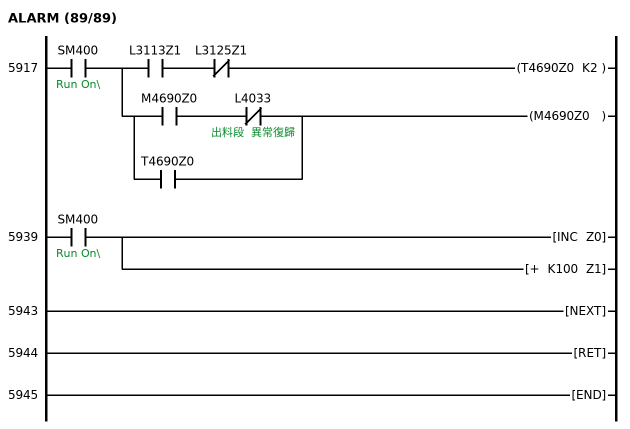
[picture p264: ladder of ALARM, rungs at steps 5917 to 5945]
5917  LD      SM400  ; Run On\
      MPS
      AND     L3113Z1
      ANI     L3125Z1
      OUT     T4690Z0 K2
      MPP
      LD      M4690Z0
      ANI     L4033  ; 出料段  異常復歸
      OR      T4690Z0
      ANB
      OUT     M4690Z0
5939  LD      SM400  ; Run On\
      INC     Z0
      +       K100 Z1
5943  NEXT
5944  RET
5945  END
END_PROGRAM

PROGRAM CCD_RB
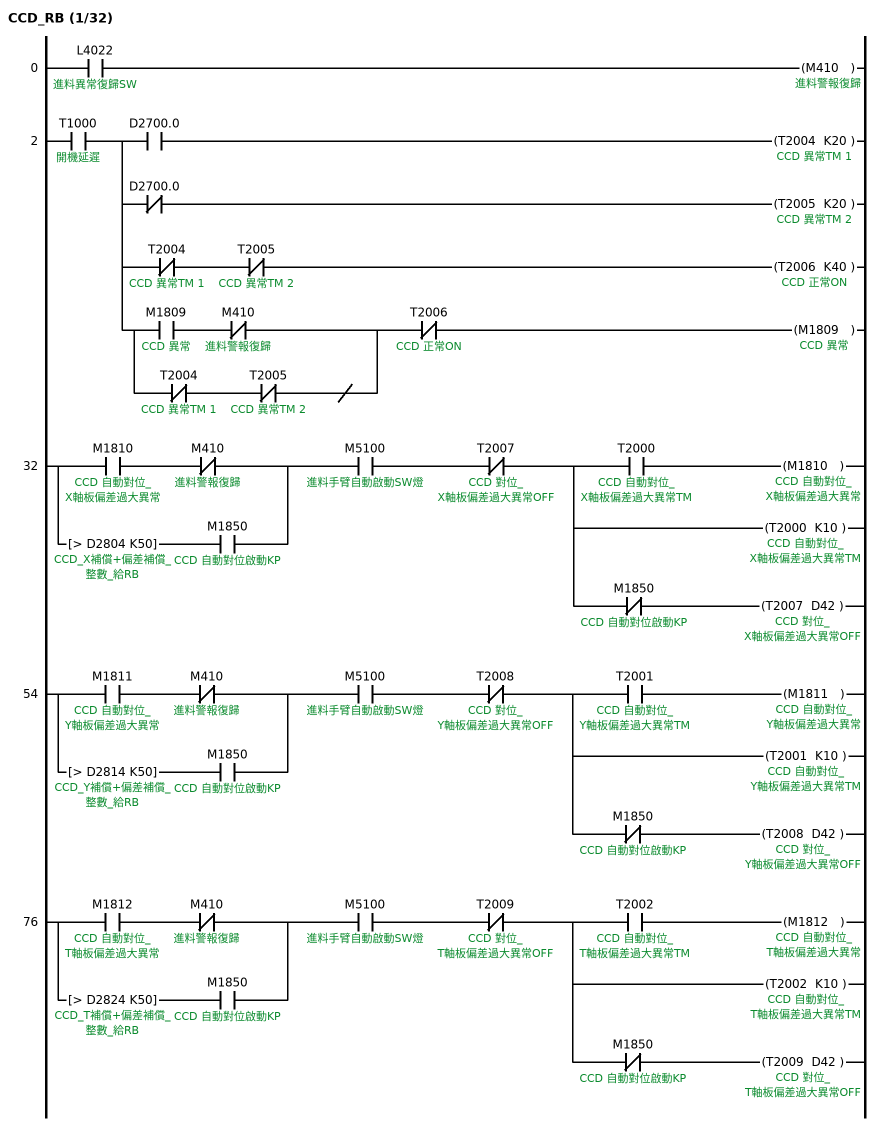
0     LD      L4022  ; 進料異常復歸SW
      OUT     M410  ; 進料警報復歸
2     LD      T1000  ; 開機延遲
      MPS
      AND     D2700.0
      OUT     T2004 K20  ; CCD 異常TM 1
      MRD
      ANI     D2700.0
      OUT     T2005 K20  ; CCD 異常TM 2
      MRD
      ANI     T2004  ; CCD 異常TM 1
      ANI     T2005  ; CCD 異常TM 2
      OUT     T2006 K40  ; CCD 正常ON
      MPP
      LD      M1809  ; CCD 異常
      ANI     M410  ; 進料警報復歸
      LDI     T2004  ; CCD 異常TM 1
      ANI     T2005  ; CCD 異常TM 2
      INV
      ORB
      ANB
      ANI     T2006  ; CCD 正常ON
      OUT     M1809  ; CCD 異常
32    LD      M1810  ; CCD 自動對位_X軸板偏差過大異常
      ANI     M410  ; 進料警報復歸
      LD>     D2804 K50  ; CCD_X補償+偏差補償_整數_給RB
      AND     M1850  ; CCD 自動對位啟動KP
      ORB
      AND     M5100  ; 進料手臂自動啟動SW燈
      ANI     T2007  ; CCD 對位_X軸板偏差過大異常OFF
      MPS
      AND     T2000  ; CCD 自動對位_X軸板偏差過大異常TM
      OUT     M1810  ; CCD 自動對位_X軸板偏差過大異常
      MPP
      OUT     T2000 K10  ; CCD 自動對位_X軸板偏差過大異常TM
      ANI     M1850  ; CCD 自動對位啟動KP
      OUT     T2007 D42  ; CCD 對位_X軸板偏差過大異常OFF
54    LD      M1811  ; CCD 自動對位_Y軸板偏差過大異常
      ANI     M410  ; 進料警報復歸
      LD>     D2814 K50  ; CCD_Y補償+偏差補償_整數_給RB
      AND     M1850  ; CCD 自動對位啟動KP
      ORB
      AND     M5100  ; 進料手臂自動啟動SW燈
      ANI     T2008  ; CCD 對位_Y軸板偏差過大異常OFF
      MPS
      AND     T2001  ; CCD 自動對位_Y軸板偏差過大異常TM
      OUT     M1811  ; CCD 自動對位_Y軸板偏差過大異常
      MPP
      OUT     T2001 K10  ; CCD 自動對位_Y軸板偏差過大異常TM
      ANI     M1850  ; CCD 自動對位啟動KP
      OUT     T2008 D42  ; CCD 對位_Y軸板偏差過大異常OFF
76    LD      M1812  ; CCD 自動對位_T軸板偏差過大異常
      ANI     M410  ; 進料警報復歸
      LD>     D2824 K50  ; CCD_T補償+偏差補償_整數_給RB
      AND     M1850  ; CCD 自動對位啟動KP
      ORB
      AND     M5100  ; 進料手臂自動啟動SW燈
      ANI     T2009  ; CCD 對位_T軸板偏差過大異常OFF
      MPS
      AND     T2002  ; CCD 自動對位_T軸板偏差過大異常TM
      OUT     M1812  ; CCD 自動對位_T軸板偏差過大異常
      MPP
      OUT     T2002 K10  ; CCD 自動對位_T軸板偏差過大異常TM
      ANI     M1850  ; CCD 自動對位啟動KP
      OUT     T2009 D42  ; CCD 對位_T軸板偏差過大異常OFF
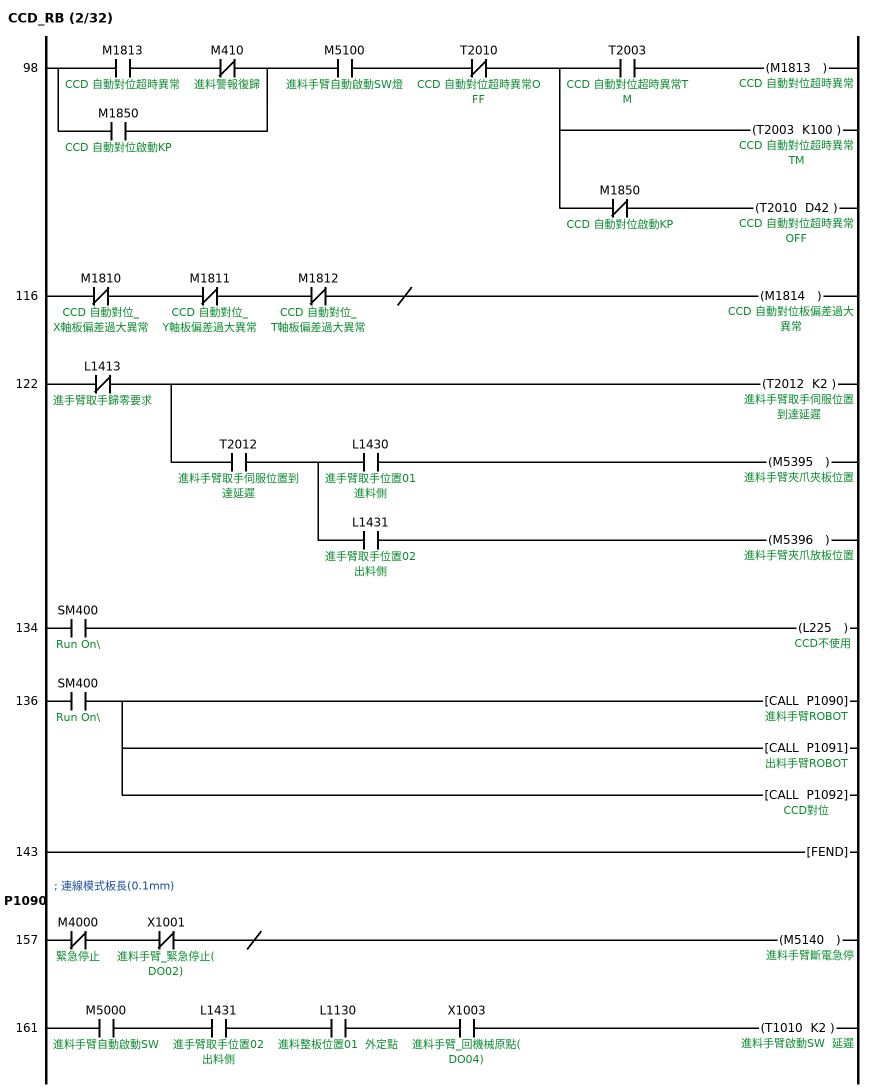
98    LD      M1813  ; CCD 自動對位超時異常
      ANI     M410  ; 進料警報復歸
      OR      M1850  ; CCD 自動對位啟動KP
      AND     M5100  ; 進料手臂自動啟動SW燈
      ANI     T2010  ; CCD 自動對位超時異常OFF
      MPS
      AND     T2003  ; CCD 自動對位超時異常TM
      OUT     M1813  ; CCD 自動對位超時異常
      MPP
      OUT     T2003 K100  ; CCD 自動對位超時異常TM
      ANI     M1850  ; CCD 自動對位啟動KP
      OUT     T2010 D42  ; CCD 自動對位超時異常OFF
116   LDI     M1810  ; CCD 自動對位_X軸板偏差過大異常
      ANI     M1811  ; CCD 自動對位_Y軸板偏差過大異常
      ANI     M1812  ; CCD 自動對位_T軸板偏差過大異常
      INV
      OUT     M1814  ; CCD 自動對位板偏差過大異常
122   LDI     L1413  ; 進手臂取手歸零要求
      OUT     T2012 K2  ; 進料手臂取手伺服位置到達延遲
      AND     T2012  ; 進料手臂取手伺服位置到達延遲
      MPS
      AND     L1430  ; 進手臂取手位置01  進料側
      OUT     M5395  ; 進料手臂夾爪夾板位置
      MPP
      AND     L1431  ; 進手臂取手位置02  出料側
      OUT     M5396  ; 進料手臂夾爪放板位置
134   LD      SM400  ; Run On\
      OUT     L225  ; CCD不使用
136   LD      SM400  ; Run On\
      CALL    P1090  ; 進料手臂ROBOT
      CALL    P1091  ; 出料手臂ROBOT
      CALL    P1092  ; CCD對位
143   FEND
; 連線模式板長(0.1mm)
      P1090
157   LDI     M4000  ; 緊急停止
      ANI     X1001  ; 進料手臂_緊急停止(DO02)
      INV
      OUT     M5140  ; 進料手臂斷電急停
161   LD      M5000  ; 進料手臂自動啟動SW
      AND     L1431  ; 進手臂取手位置02  出料側
      AND     L1130  ; 進料整板位置01  外定點
      AND     X1003  ; 進料手臂_回機械原點(DO04)
      OUT     T1010 K2  ; 進料手臂啟動SW  延遲
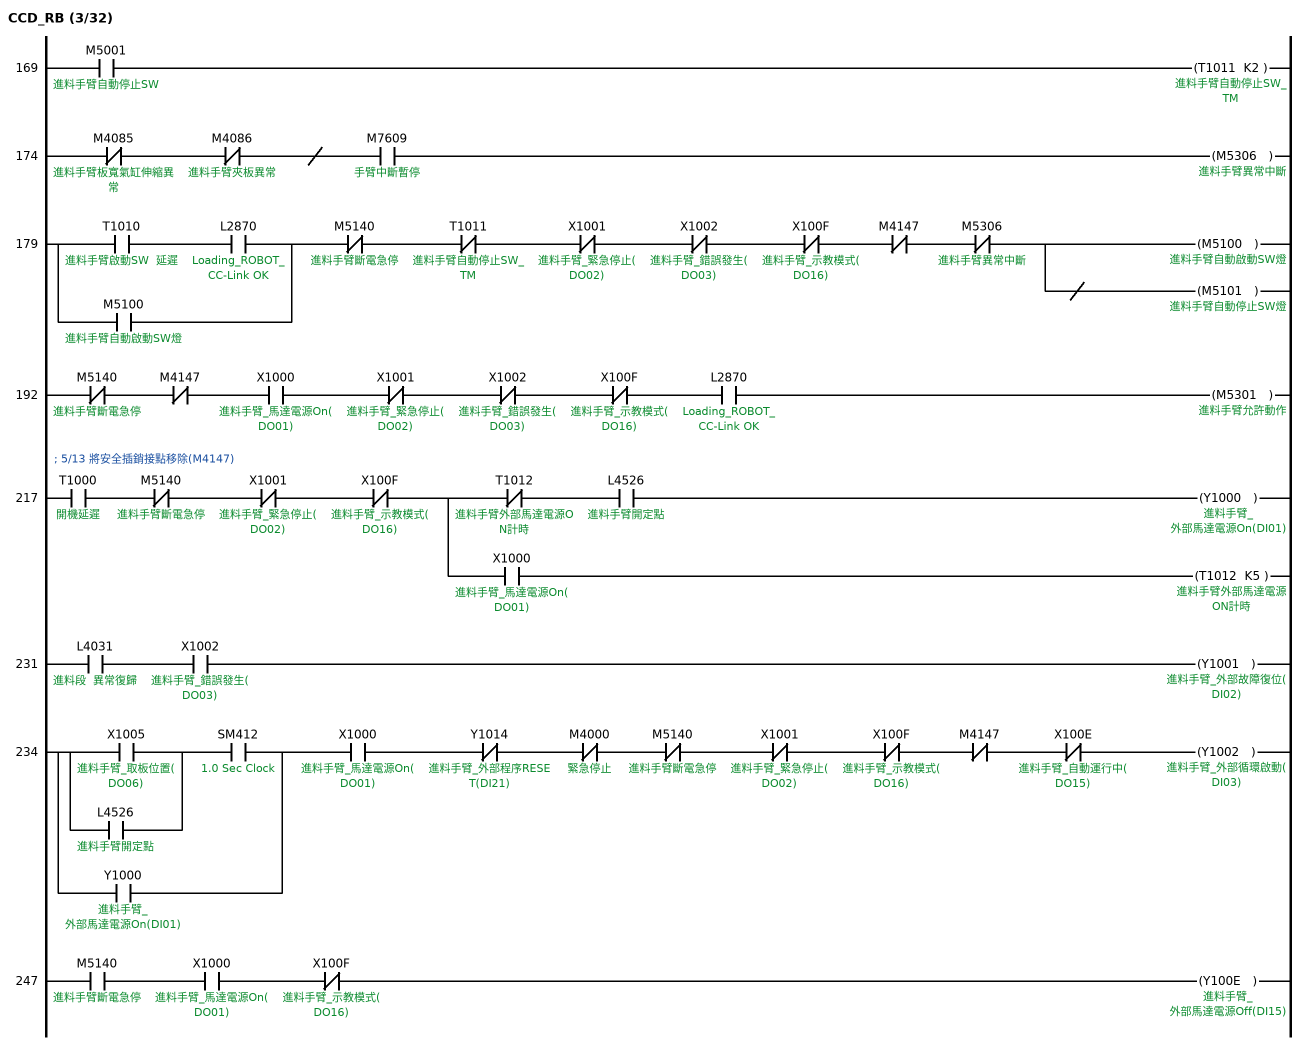
169   LD      M5001  ; 進料手臂自動停止SW
      OUT     T1011 K2  ; 進料手臂自動停止SW_TM
174   LDI     M4085  ; 進料手臂板寬氣缸伸縮異常
      ANI     M4086  ; 進料手臂夾板異常
      INV
      AND     M7609  ; 手臂中斷暫停
      OUT     M5306  ; 進料手臂異常中斷
179   LD      T1010  ; 進料手臂啟動SW  延遲
      AND     L2870  ; Loading_ROBOT_  CC-Link OK
      OR      M5100  ; 進料手臂自動啟動SW燈
      ANI     M5140  ; 進料手臂斷電急停
      ANI     T1011  ; 進料手臂自動停止SW_TM
      ANI     X1001  ; 進料手臂_緊急停止(DO02)
      ANI     X1002  ; 進料手臂_錯誤發生(DO03)
      ANI     X100F  ; 進料手臂_示教模式(DO16)
      ANI     M4147
      ANI     M5306  ; 進料手臂異常中斷
      OUT     M5100  ; 進料手臂自動啟動SW燈
      INV
      OUT     M5101  ; 進料手臂自動停止SW燈
192   LDI     M5140  ; 進料手臂斷電急停
      ANI     M4147
      AND     X1000  ; 進料手臂_馬達電源On(DO01)
      ANI     X1001  ; 進料手臂_緊急停止(DO02)
      ANI     X1002  ; 進料手臂_錯誤發生(DO03)
      ANI     X100F  ; 進料手臂_示教模式(DO16)
      AND     L2870  ; Loading_ROBOT_  CC-Link OK
      OUT     M5301  ; 進料手臂允許動作
; 5/13 將安全插銷接點移除(M4147)
217   LD      T1000  ; 開機延遲
      ANI     M5140  ; 進料手臂斷電急停
      ANI     X1001  ; 進料手臂_緊急停止(DO02)
      ANI     X100F  ; 進料手臂_示教模式(DO16)
      MPS
      ANI     T1012  ; 進料手臂外部馬達電源ON計時
      AND     L4526  ; 進料手臂開定點
      OUT     Y1000  ; 進料手臂_外部馬達電源On(DI01)
      MPP
      AND     X1000  ; 進料手臂_馬達電源On(DO01)
      OUT     T1012 K5  ; 進料手臂外部馬達電源ON計時
231   LD      L4031  ; 進料段  異常復歸
      AND     X1002  ; 進料手臂_錯誤發生(DO03)
      OUT     Y1001  ; 進料手臂_外部故障復位(DI02)
234   LD      X1005  ; 進料手臂_取板位置(DO06)
      OR      L4526  ; 進料手臂開定點
      AND     SM412  ; 1.0 Sec Clock
      OR      Y1000  ; 進料手臂_外部馬達電源On(DI01)
      AND     X1000  ; 進料手臂_馬達電源On(DO01)
      ANI     Y1014  ; 進料手臂_外部程序RESET(DI21)
      ANI     M4000  ; 緊急停止
      ANI     M5140  ; 進料手臂斷電急停
      ANI     X1001  ; 進料手臂_緊急停止(DO02)
      ANI     X100F  ; 進料手臂_示教模式(DO16)
      ANI     M4147
      ANI     X100E  ; 進料手臂_自動運行中(DO15)
      OUT     Y1002  ; 進料手臂_外部循環啟動(DI03)
247   LD      M5140  ; 進料手臂斷電急停
      AND     X1000  ; 進料手臂_馬達電源On(DO01)
      ANI     X100F  ; 進料手臂_示教模式(DO16)
      OUT     Y100E  ; 進料手臂_外部馬達電源Off(DI15)
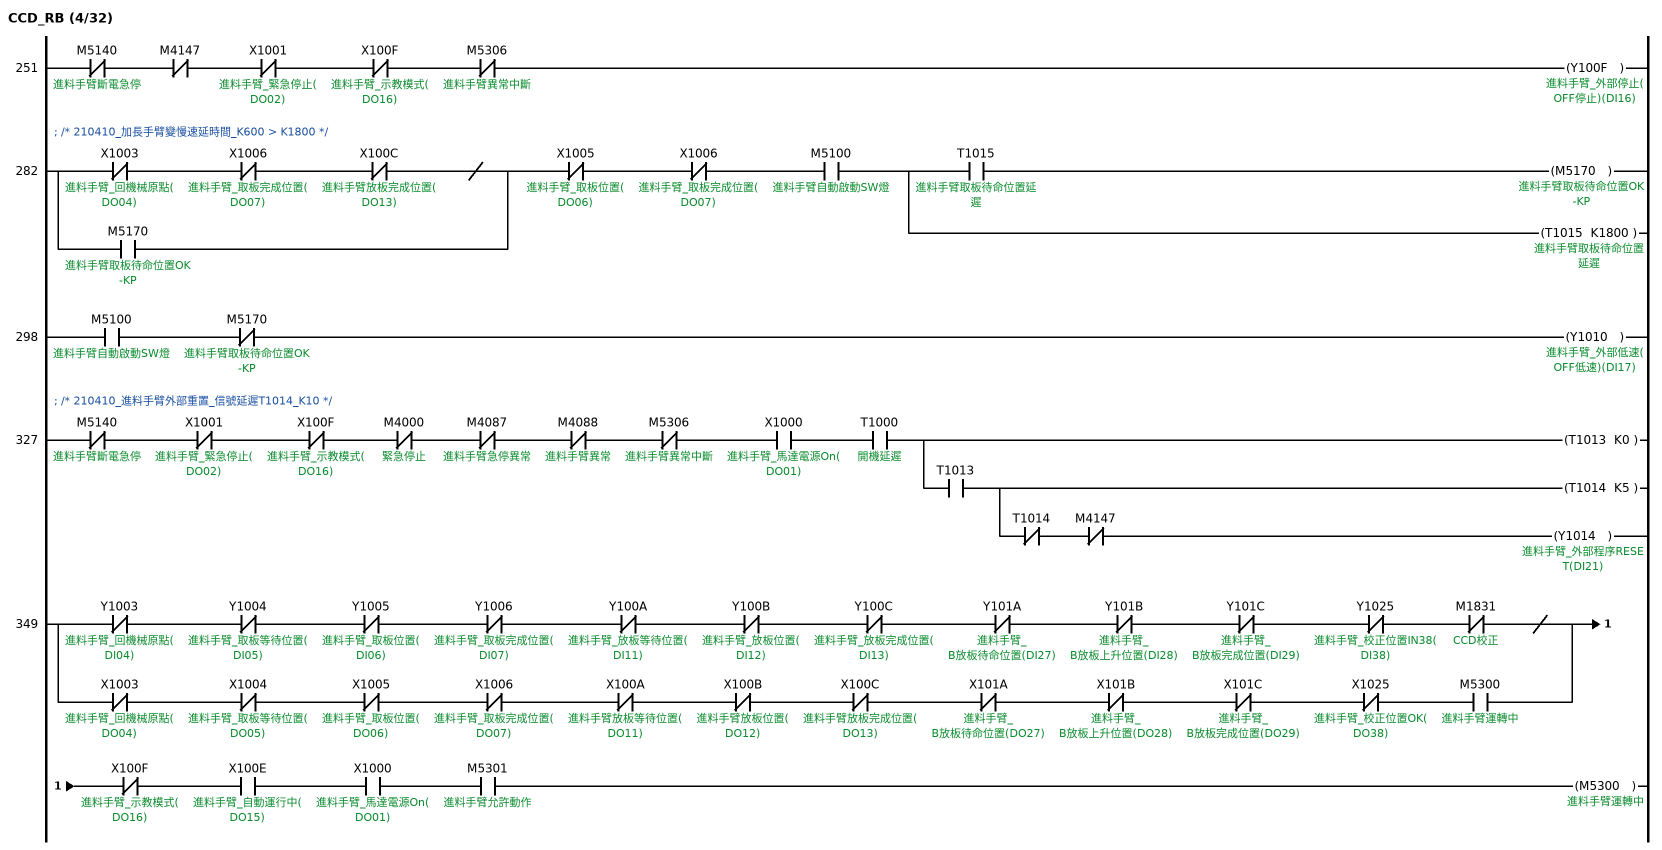
251   LDI     M5140  ; 進料手臂斷電急停
      ANI     M4147
      ANI     X1001  ; 進料手臂_緊急停止(DO02)
      ANI     X100F  ; 進料手臂_示教模式(DO16)
      ANI     M5306  ; 進料手臂異常中斷
      OUT     Y100F  ; 進料手臂_外部停止(OFF停止)(DI16)
; /* 210410_加長手臂變慢速延時間_K600 > K1800 */
282   LDI     X1003  ; 進料手臂_回機械原點(DO04)
      ANI     X1006  ; 進料手臂_取板完成位置(DO07)
      ANI     X100C  ; 進料手臂放板完成位置(DO13)
      INV
      OR      M5170  ; 進料手臂取板待命位置OK-KP
      ANI     X1005  ; 進料手臂_取板位置(DO06)
      ANI     X1006  ; 進料手臂_取板完成位置(DO07)
      AND     M5100  ; 進料手臂自動啟動SW燈
      MPS
      AND     T1015  ; 進料手臂取板待命位置延遲
      OUT     M5170  ; 進料手臂取板待命位置OK-KP
      MPP
      OUT     T1015 K1800  ; 進料手臂取板待命位置延遲
298   LD      M5100  ; 進料手臂自動啟動SW燈
      ANI     M5170  ; 進料手臂取板待命位置OK-KP
      OUT     Y1010  ; 進料手臂_外部低速(OFF低速)(DI17)
; /* 210410_進料手臂外部重置_信號延遲T1014_K10 */
327   LDI     M5140  ; 進料手臂斷電急停
      ANI     X1001  ; 進料手臂_緊急停止(DO02)
      ANI     X100F  ; 進料手臂_示教模式(DO16)
      ANI     M4000  ; 緊急停止
      ANI     M4087  ; 進料手臂急停異常
      ANI     M4088  ; 進料手臂異常
      ANI     M5306  ; 進料手臂異常中斷
      AND     X1000  ; 進料手臂_馬達電源On(DO01)
      AND     T1000  ; 開機延遲
      OUT     T1013 K0
      AND     T1013
      OUT     T1014 K5
      ANI     T1014
      ANI     M4147
      OUT     Y1014  ; 進料手臂_外部程序RESET(DI21)
349   LDI     Y1003  ; 進料手臂_回機械原點(DI04)
      ANI     Y1004  ; 進料手臂_取板等待位置(DI05)
      ANI     Y1005  ; 進料手臂_取板位置(DI06)
      ANI     Y1006  ; 進料手臂_取板完成位置(DI07)
      ANI     Y100A  ; 進料手臂_放板等待位置(DI11)
      ANI     Y100B  ; 進料手臂_放板位置(DI12)
      ANI     Y100C  ; 進料手臂_放板完成位置(DI13)
      ANI     Y101A  ; 進料手臂_B放板待命位置(DI27)
      ANI     Y101B  ; 進料手臂_B放板上升位置(DI28)
      ANI     Y101C  ; 進料手臂_B放板完成位置(DI29)
      ANI     Y1025  ; 進料手臂_校正位置IN38(DI38)
      ANI     M1831  ; CCD校正
      INV
      LDI     X1003  ; 進料手臂_回機械原點(DO04)
      ANI     X1004  ; 進料手臂_取板等待位置(DO05)
      ANI     X1005  ; 進料手臂_取板位置(DO06)
      ANI     X1006  ; 進料手臂_取板完成位置(DO07)
      ANI     X100A  ; 進料手臂放板等待位置(DO11)
      ANI     X100B  ; 進料手臂放板位置(DO12)
      ANI     X100C  ; 進料手臂放板完成位置(DO13)
      ANI     X101A  ; 進料手臂_B放板待命位置(DO27)
      ANI     X101B  ; 進料手臂_B放板上升位置(DO28)
      ANI     X101C  ; 進料手臂_B放板完成位置(DO29)
      ANI     X1025  ; 進料手臂_校正位置OK(DO38)
      AND     M5300  ; 進料手臂運轉中
      ORB
      ANI     X100F  ; 進料手臂_示教模式(DO16)
      AND     X100E  ; 進料手臂_自動運行中(DO15)
      AND     X1000  ; 進料手臂_馬達電源On(DO01)
      AND     M5301  ; 進料手臂允許動作
      OUT     M5300  ; 進料手臂運轉中
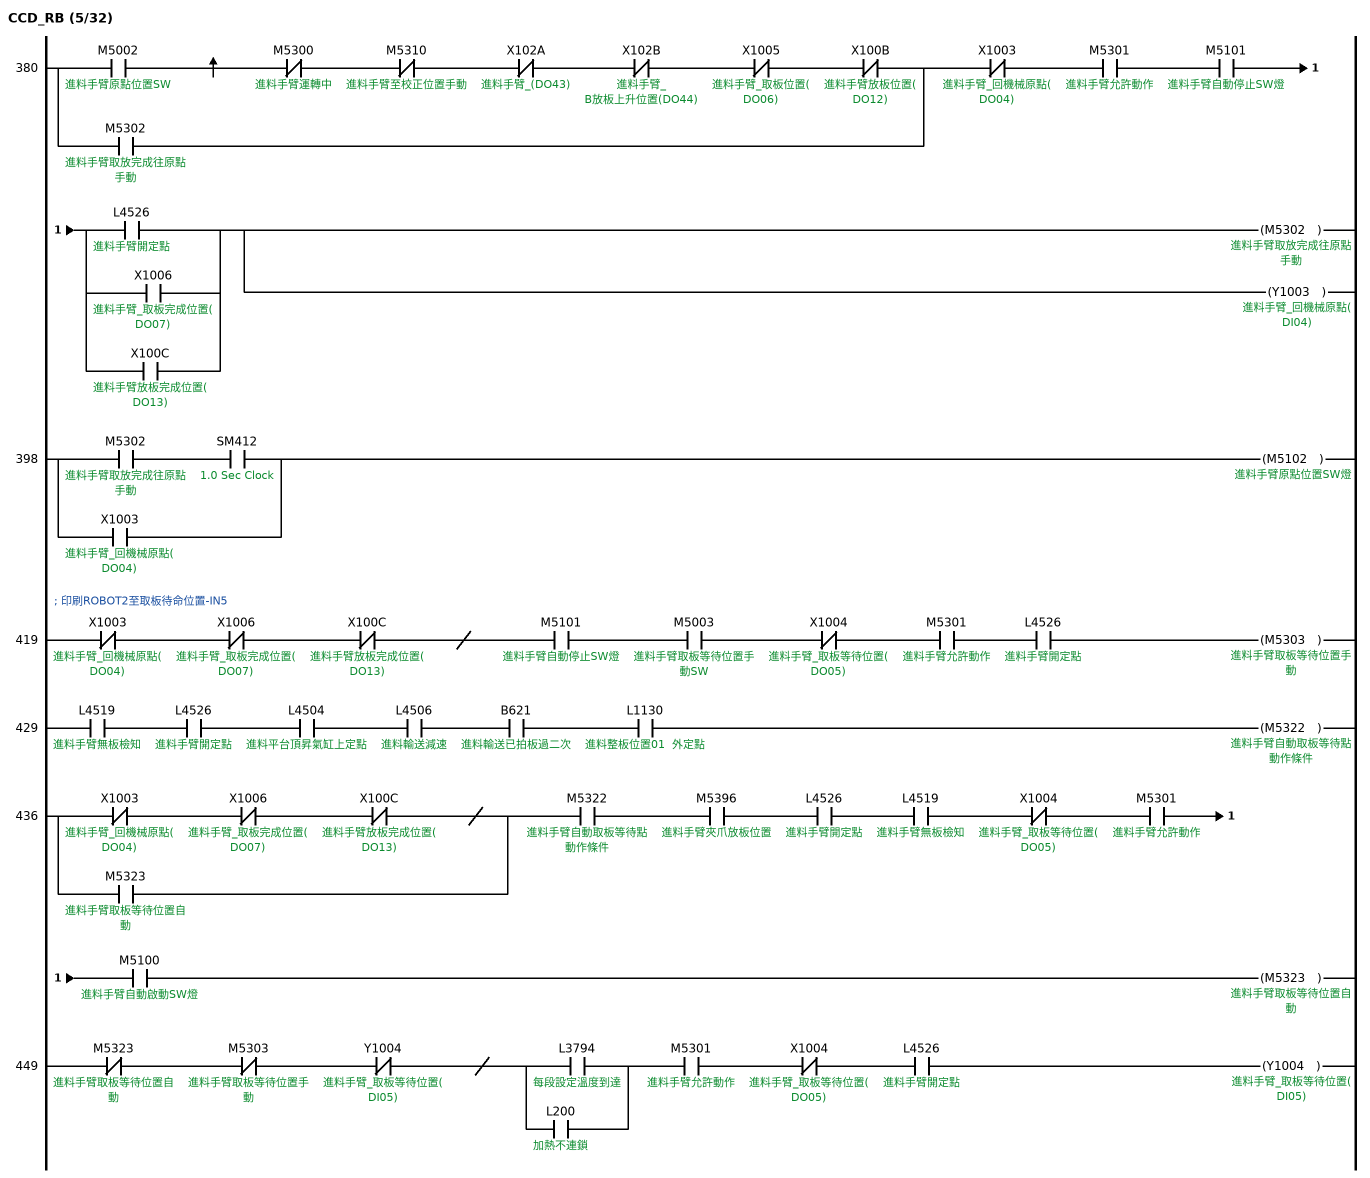
380   LD      M5002  ; 進料手臂原點位置SW
      MEP
      ANI     M5300  ; 進料手臂運轉中
      ANI     M5310  ; 進料手臂至校正位置手動
      ANI     X102A  ; 進料手臂_(DO43)
      ANI     X102B  ; 進料手臂_B放板上升位置(DO44)
      ANI     X1005  ; 進料手臂_取板位置(DO06)
      ANI     X100B  ; 進料手臂放板位置(DO12)
      OR      M5302  ; 進料手臂取放完成往原點手動
      ANI     X1003  ; 進料手臂_回機械原點(DO04)
      AND     M5301  ; 進料手臂允許動作
      AND     M5101  ; 進料手臂自動停止SW燈
      LD      L4526  ; 進料手臂開定點
      OR      X1006  ; 進料手臂_取板完成位置(DO07)
      OR      X100C  ; 進料手臂放板完成位置(DO13)
      ANB
      OUT     M5302  ; 進料手臂取放完成往原點手動
      OUT     Y1003  ; 進料手臂_回機械原點(DI04)
398   LD      M5302  ; 進料手臂取放完成往原點手動
      AND     SM412  ; 1.0 Sec Clock
      OR      X1003  ; 進料手臂_回機械原點(DO04)
      OUT     M5102  ; 進料手臂原點位置SW燈
; 印刷ROBOT2至取板待命位置-IN5
419   LDI     X1003  ; 進料手臂_回機械原點(DO04)
      ANI     X1006  ; 進料手臂_取板完成位置(DO07)
      ANI     X100C  ; 進料手臂放板完成位置(DO13)
      INV
      AND     M5101  ; 進料手臂自動停止SW燈
      AND     M5003  ; 進料手臂取板等待位置手動SW
      ANI     X1004  ; 進料手臂_取板等待位置(DO05)
      AND     M5301  ; 進料手臂允許動作
      AND     L4526  ; 進料手臂開定點
      OUT     M5303  ; 進料手臂取板等待位置手動
429   LD      L4519  ; 進料手臂無板檢知
      AND     L4526  ; 進料手臂開定點
      AND     L4504  ; 進料平台頂昇氣缸上定點
      AND     L4506  ; 進料輸送減速
      AND     B621  ; 進料輸送已拍板過二次
      AND     L1130  ; 進料整板位置01  外定點
      OUT     M5322  ; 進料手臂自動取板等待點動作條件
436   LDI     X1003  ; 進料手臂_回機械原點(DO04)
      ANI     X1006  ; 進料手臂_取板完成位置(DO07)
      ANI     X100C  ; 進料手臂放板完成位置(DO13)
      INV
      OR      M5323  ; 進料手臂取板等待位置自動
      AND     M5322  ; 進料手臂自動取板等待點動作條件
      AND     M5396  ; 進料手臂夾爪放板位置
      AND     L4526  ; 進料手臂開定點
      AND     L4519  ; 進料手臂無板檢知
      ANI     X1004  ; 進料手臂_取板等待位置(DO05)
      AND     M5301  ; 進料手臂允許動作
      AND     M5100  ; 進料手臂自動啟動SW燈
      OUT     M5323  ; 進料手臂取板等待位置自動
449   LDI     M5323  ; 進料手臂取板等待位置自動
      ANI     M5303  ; 進料手臂取板等待位置手動
      ANI     Y1004  ; 進料手臂_取板等待位置(DI05)
      INV
      LD      L3794  ; 每段設定溫度到達
      OR      L200  ; 加熱不連鎖
      ANB
      AND     M5301  ; 進料手臂允許動作
      ANI     X1004  ; 進料手臂_取板等待位置(DO05)
      AND     L4526  ; 進料手臂開定點
      OUT     Y1004  ; 進料手臂_取板等待位置(DI05)
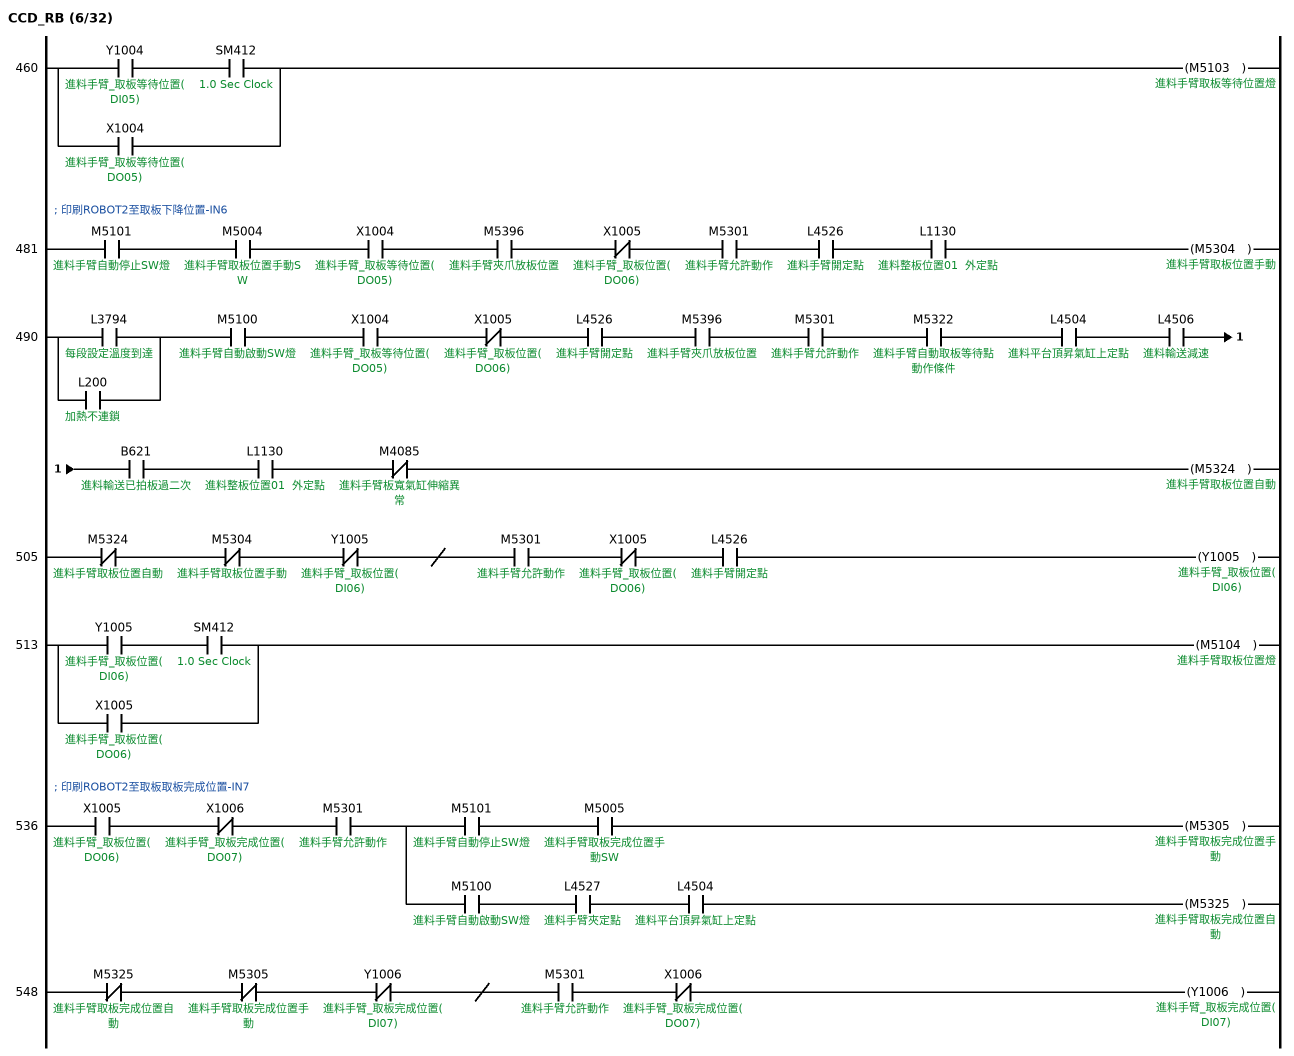
460   LD      Y1004  ; 進料手臂_取板等待位置(DI05)
      AND     SM412  ; 1.0 Sec Clock
      OR      X1004  ; 進料手臂_取板等待位置(DO05)
      OUT     M5103  ; 進料手臂取板等待位置燈
; 印刷ROBOT2至取板下降位置-IN6
481   LD      M5101  ; 進料手臂自動停止SW燈
      AND     M5004  ; 進料手臂取板位置手動SW
      AND     X1004  ; 進料手臂_取板等待位置(DO05)
      AND     M5396  ; 進料手臂夾爪放板位置
      ANI     X1005  ; 進料手臂_取板位置(DO06)
      AND     M5301  ; 進料手臂允許動作
      AND     L4526  ; 進料手臂開定點
      AND     L1130  ; 進料整板位置01  外定點
      OUT     M5304  ; 進料手臂取板位置手動
490   LD      L3794  ; 每段設定溫度到達
      OR      L200  ; 加熱不連鎖
      AND     M5100  ; 進料手臂自動啟動SW燈
      AND     X1004  ; 進料手臂_取板等待位置(DO05)
      ANI     X1005  ; 進料手臂_取板位置(DO06)
      AND     L4526  ; 進料手臂開定點
      AND     M5396  ; 進料手臂夾爪放板位置
      AND     M5301  ; 進料手臂允許動作
      AND     M5322  ; 進料手臂自動取板等待點動作條件
      AND     L4504  ; 進料平台頂昇氣缸上定點
      AND     L4506  ; 進料輸送減速
      AND     B621  ; 進料輸送已拍板過二次
      AND     L1130  ; 進料整板位置01  外定點
      ANI     M4085  ; 進料手臂板寬氣缸伸縮異常
      OUT     M5324  ; 進料手臂取板位置自動
505   LDI     M5324  ; 進料手臂取板位置自動
      ANI     M5304  ; 進料手臂取板位置手動
      ANI     Y1005  ; 進料手臂_取板位置(DI06)
      INV
      AND     M5301  ; 進料手臂允許動作
      ANI     X1005  ; 進料手臂_取板位置(DO06)
      AND     L4526  ; 進料手臂開定點
      OUT     Y1005  ; 進料手臂_取板位置(DI06)
513   LD      Y1005  ; 進料手臂_取板位置(DI06)
      AND     SM412  ; 1.0 Sec Clock
      OR      X1005  ; 進料手臂_取板位置(DO06)
      OUT     M5104  ; 進料手臂取板位置燈
; 印刷ROBOT2至取板取板完成位置-IN7
536   LD      X1005  ; 進料手臂_取板位置(DO06)
      ANI     X1006  ; 進料手臂_取板完成位置(DO07)
      AND     M5301  ; 進料手臂允許動作
      MPS
      AND     M5101  ; 進料手臂自動停止SW燈
      AND     M5005  ; 進料手臂取板完成位置手動SW
      OUT     M5305  ; 進料手臂取板完成位置手動
      MPP
      AND     M5100  ; 進料手臂自動啟動SW燈
      AND     L4527  ; 進料手臂夾定點
      AND     L4504  ; 進料平台頂昇氣缸上定點
      OUT     M5325  ; 進料手臂取板完成位置自動
548   LDI     M5325  ; 進料手臂取板完成位置自動
      ANI     M5305  ; 進料手臂取板完成位置手動
      ANI     Y1006  ; 進料手臂_取板完成位置(DI07)
      INV
      AND     M5301  ; 進料手臂允許動作
      ANI     X1006  ; 進料手臂_取板完成位置(DO07)
      OUT     Y1006  ; 進料手臂_取板完成位置(DI07)
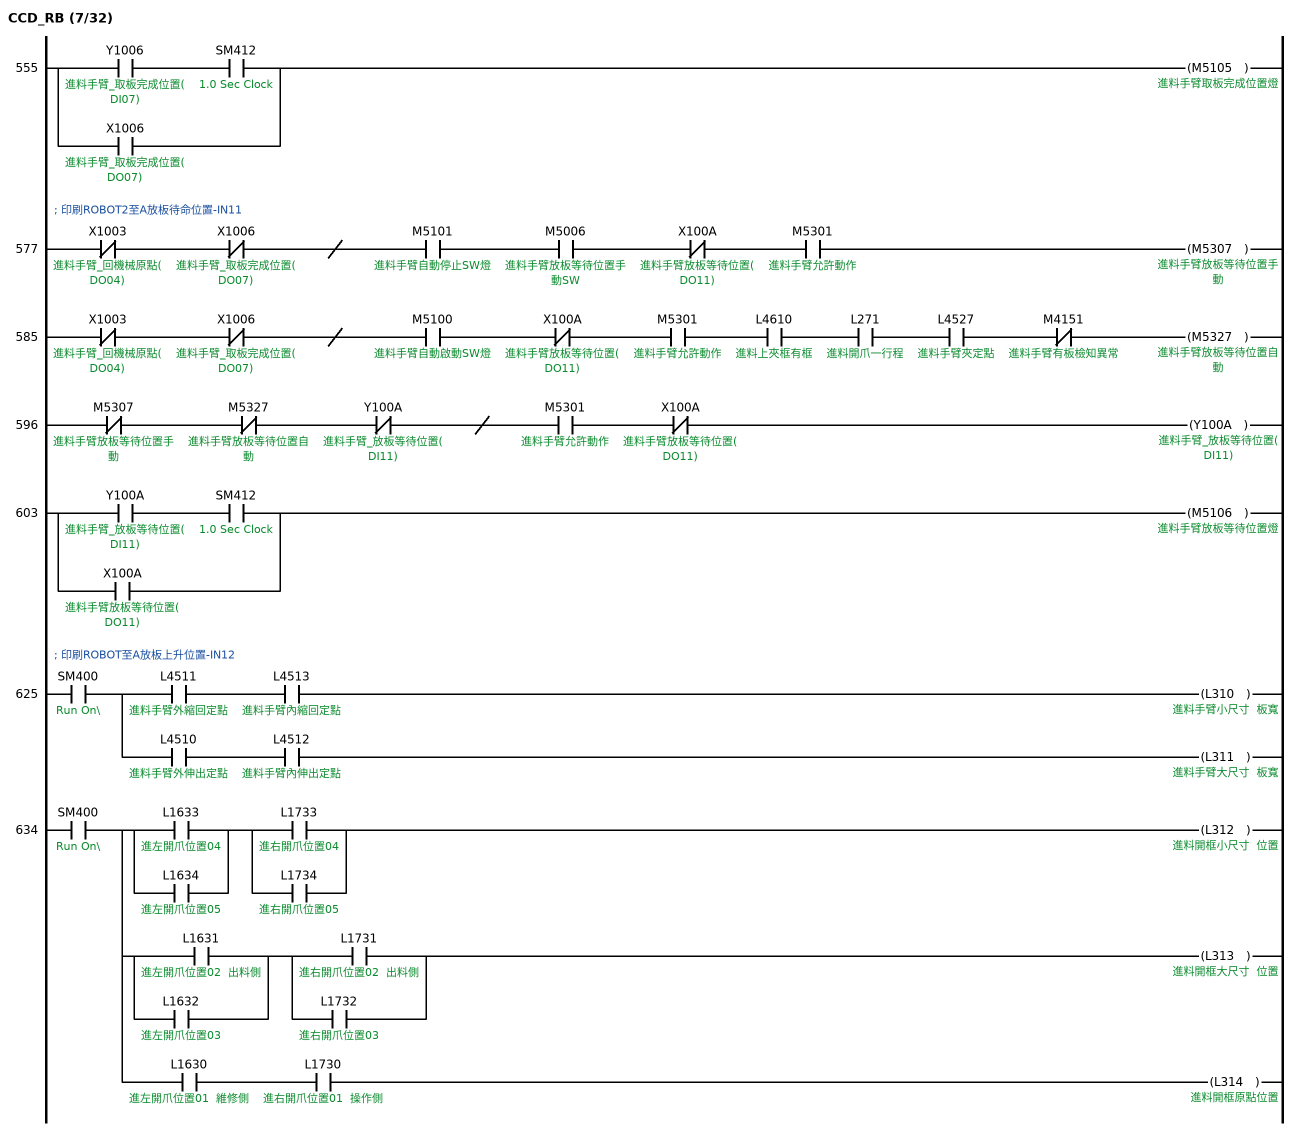
555   LD      Y1006  ; 進料手臂_取板完成位置(DI07)
      AND     SM412  ; 1.0 Sec Clock
      OR      X1006  ; 進料手臂_取板完成位置(DO07)
      OUT     M5105  ; 進料手臂取板完成位置燈
; 印刷ROBOT2至A放板待命位置-IN11
577   LDI     X1003  ; 進料手臂_回機械原點(DO04)
      ANI     X1006  ; 進料手臂_取板完成位置(DO07)
      INV
      AND     M5101  ; 進料手臂自動停止SW燈
      AND     M5006  ; 進料手臂放板等待位置手動SW
      ANI     X100A  ; 進料手臂放板等待位置(DO11)
      AND     M5301  ; 進料手臂允許動作
      OUT     M5307  ; 進料手臂放板等待位置手動
585   LDI     X1003  ; 進料手臂_回機械原點(DO04)
      ANI     X1006  ; 進料手臂_取板完成位置(DO07)
      INV
      AND     M5100  ; 進料手臂自動啟動SW燈
      ANI     X100A  ; 進料手臂放板等待位置(DO11)
      AND     M5301  ; 進料手臂允許動作
      AND     L4610  ; 進料上夾框有框
      AND     L271  ; 進料開爪一行程
      AND     L4527  ; 進料手臂夾定點
      ANI     M4151  ; 進料手臂有板檢知異常
      OUT     M5327  ; 進料手臂放板等待位置自動
596   LDI     M5307  ; 進料手臂放板等待位置手動
      ANI     M5327  ; 進料手臂放板等待位置自動
      ANI     Y100A  ; 進料手臂_放板等待位置(DI11)
      INV
      AND     M5301  ; 進料手臂允許動作
      ANI     X100A  ; 進料手臂放板等待位置(DO11)
      OUT     Y100A  ; 進料手臂_放板等待位置(DI11)
603   LD      Y100A  ; 進料手臂_放板等待位置(DI11)
      AND     SM412  ; 1.0 Sec Clock
      OR      X100A  ; 進料手臂放板等待位置(DO11)
      OUT     M5106  ; 進料手臂放板等待位置燈
; 印刷ROBOT至A放板上升位置-IN12
625   LD      SM400  ; Run On\
      MPS
      AND     L4511  ; 進料手臂外縮回定點
      AND     L4513  ; 進料手臂內縮回定點
      OUT     L310  ; 進料手臂小尺寸  板寬
      MPP
      AND     L4510  ; 進料手臂外伸出定點
      AND     L4512  ; 進料手臂內伸出定點
      OUT     L311  ; 進料手臂大尺寸  板寬
634   LD      SM400  ; Run On\
      MPS
      LD      L1633  ; 進左開爪位置04
      OR      L1634  ; 進左開爪位置05
      ANB
      LD      L1733  ; 進右開爪位置04
      OR      L1734  ; 進右開爪位置05
      ANB
      OUT     L312  ; 進料開框小尺寸  位置
      MRD
      LD      L1631  ; 進左開爪位置02  出料側
      OR      L1632  ; 進左開爪位置03
      ANB
      LD      L1731  ; 進右開爪位置02  出料側
      OR      L1732  ; 進右開爪位置03
      ANB
      OUT     L313  ; 進料開框大尺寸  位置
      MPP
      AND     L1630  ; 進左開爪位置01  維修側
      AND     L1730  ; 進右開爪位置01  操作側
      OUT     L314  ; 進料開框原點位置
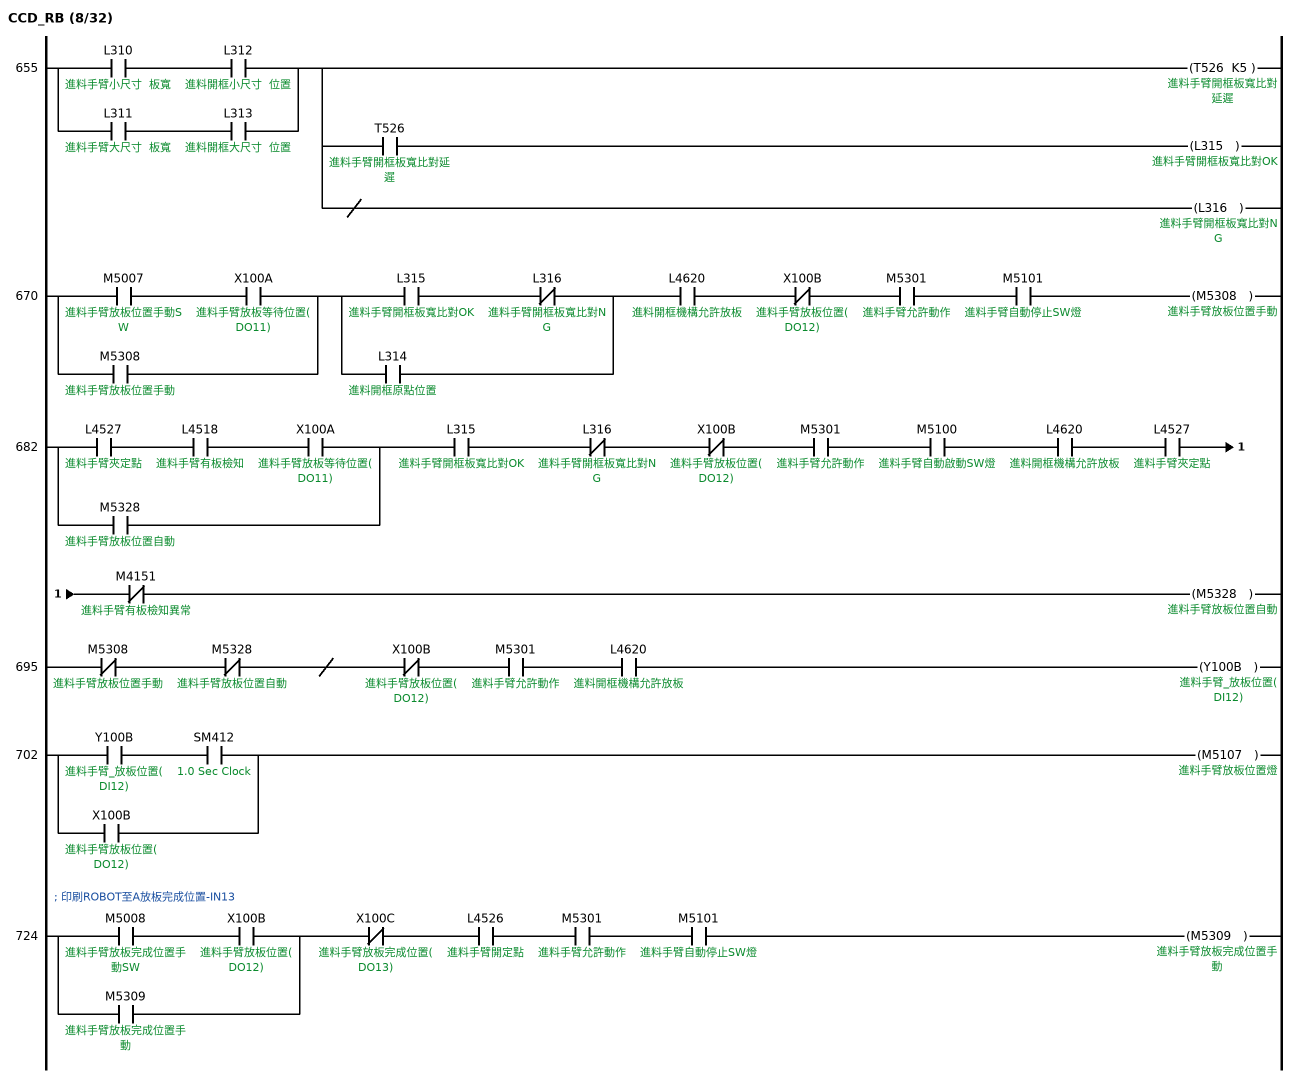
655   LD      L310  ; 進料手臂小尺寸  板寬
      AND     L312  ; 進料開框小尺寸  位置
      LD      L311  ; 進料手臂大尺寸  板寬
      AND     L313  ; 進料開框大尺寸  位置
      ORB
      OUT     T526 K5  ; 進料手臂開框板寬比對延遲
      MPS
      AND     T526  ; 進料手臂開框板寬比對延遲
      OUT     L315  ; 進料手臂開框板寬比對OK
      MPP
      INV
      OUT     L316  ; 進料手臂開框板寬比對NG
670   LD      M5007  ; 進料手臂放板位置手動SW
      AND     X100A  ; 進料手臂放板等待位置(DO11)
      OR      M5308  ; 進料手臂放板位置手動
      LD      L315  ; 進料手臂開框板寬比對OK
      ANI     L316  ; 進料手臂開框板寬比對NG
      OR      L314  ; 進料開框原點位置
      ANB
      AND     L4620  ; 進料開框機構允許放板
      ANI     X100B  ; 進料手臂放板位置(DO12)
      AND     M5301  ; 進料手臂允許動作
      AND     M5101  ; 進料手臂自動停止SW燈
      OUT     M5308  ; 進料手臂放板位置手動
682   LD      L4527  ; 進料手臂夾定點
      AND     L4518  ; 進料手臂有板檢知
      AND     X100A  ; 進料手臂放板等待位置(DO11)
      OR      M5328  ; 進料手臂放板位置自動
      AND     L315  ; 進料手臂開框板寬比對OK
      ANI     L316  ; 進料手臂開框板寬比對NG
      ANI     X100B  ; 進料手臂放板位置(DO12)
      AND     M5301  ; 進料手臂允許動作
      AND     M5100  ; 進料手臂自動啟動SW燈
      AND     L4620  ; 進料開框機構允許放板
      AND     L4527  ; 進料手臂夾定點
      ANI     M4151  ; 進料手臂有板檢知異常
      OUT     M5328  ; 進料手臂放板位置自動
695   LDI     M5308  ; 進料手臂放板位置手動
      ANI     M5328  ; 進料手臂放板位置自動
      INV
      ANI     X100B  ; 進料手臂放板位置(DO12)
      AND     M5301  ; 進料手臂允許動作
      AND     L4620  ; 進料開框機構允許放板
      OUT     Y100B  ; 進料手臂_放板位置(DI12)
702   LD      Y100B  ; 進料手臂_放板位置(DI12)
      AND     SM412  ; 1.0 Sec Clock
      OR      X100B  ; 進料手臂放板位置(DO12)
      OUT     M5107  ; 進料手臂放板位置燈
; 印刷ROBOT至A放板完成位置-IN13
724   LD      M5008  ; 進料手臂放板完成位置手動SW
      AND     X100B  ; 進料手臂放板位置(DO12)
      OR      M5309  ; 進料手臂放板完成位置手動
      ANI     X100C  ; 進料手臂放板完成位置(DO13)
      AND     L4526  ; 進料手臂開定點
      AND     M5301  ; 進料手臂允許動作
      AND     M5101  ; 進料手臂自動停止SW燈
      OUT     M5309  ; 進料手臂放板完成位置手動
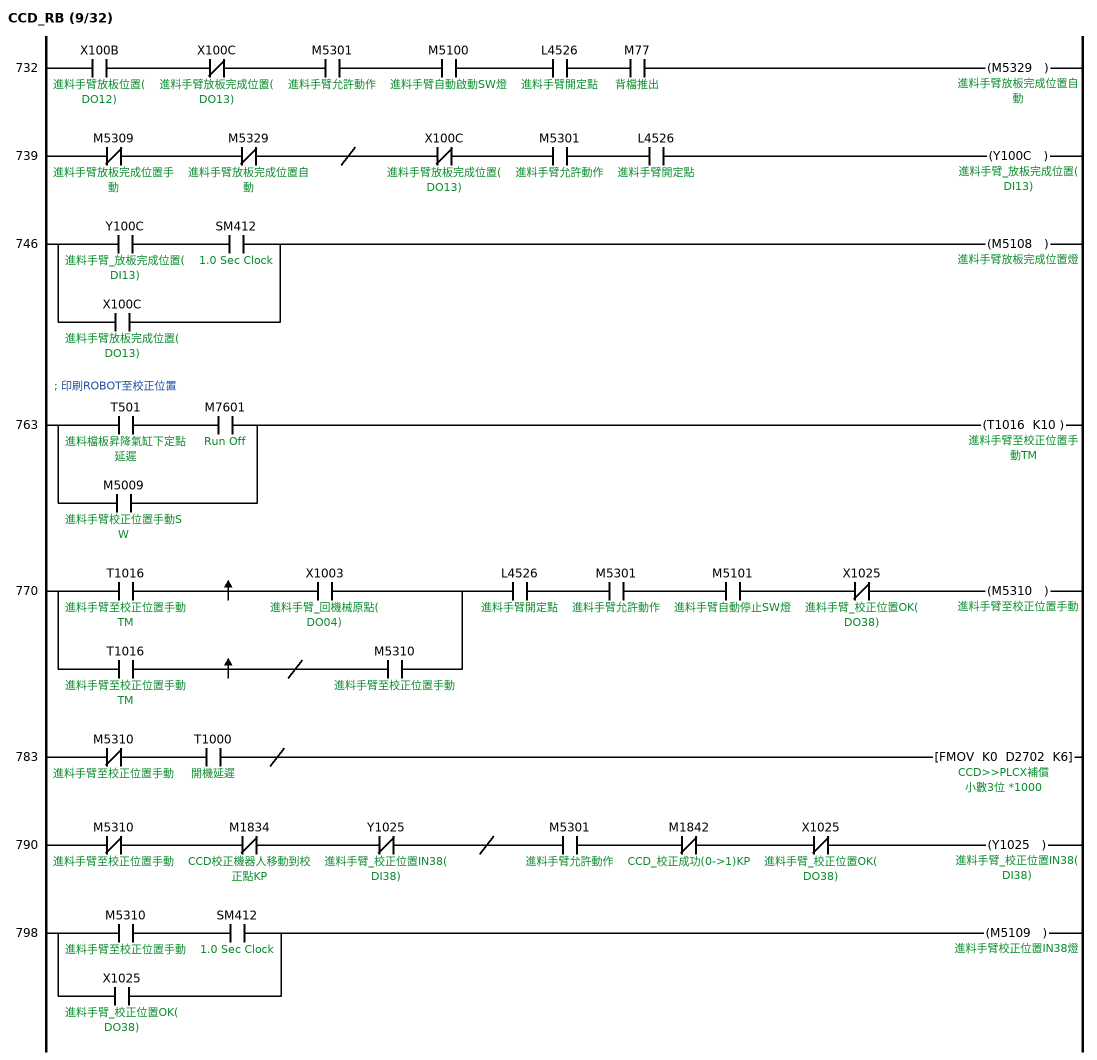
732   LD      X100B  ; 進料手臂放板位置(DO12)
      ANI     X100C  ; 進料手臂放板完成位置(DO13)
      AND     M5301  ; 進料手臂允許動作
      AND     M5100  ; 進料手臂自動啟動SW燈
      AND     L4526  ; 進料手臂開定點
      AND     M77  ; 背檔推出
      OUT     M5329  ; 進料手臂放板完成位置自動
739   LDI     M5309  ; 進料手臂放板完成位置手動
      ANI     M5329  ; 進料手臂放板完成位置自動
      INV
      ANI     X100C  ; 進料手臂放板完成位置(DO13)
      AND     M5301  ; 進料手臂允許動作
      AND     L4526  ; 進料手臂開定點
      OUT     Y100C  ; 進料手臂_放板完成位置(DI13)
746   LD      Y100C  ; 進料手臂_放板完成位置(DI13)
      AND     SM412  ; 1.0 Sec Clock
      OR      X100C  ; 進料手臂放板完成位置(DO13)
      OUT     M5108  ; 進料手臂放板完成位置燈
; 印刷ROBOT至校正位置
763   LD      T501  ; 進料檔板昇降氣缸下定點延遲
      AND     M7601  ; Run Off
      OR      M5009  ; 進料手臂校正位置手動SW
      OUT     T1016 K10  ; 進料手臂至校正位置手動TM
770   LD      T1016  ; 進料手臂至校正位置手動TM
      MEP
      AND     X1003  ; 進料手臂_回機械原點(DO04)
      LD      T1016  ; 進料手臂至校正位置手動TM
      MEP
      INV
      AND     M5310  ; 進料手臂至校正位置手動
      ORB
      AND     L4526  ; 進料手臂開定點
      AND     M5301  ; 進料手臂允許動作
      AND     M5101  ; 進料手臂自動停止SW燈
      ANI     X1025  ; 進料手臂_校正位置OK(DO38)
      OUT     M5310  ; 進料手臂至校正位置手動
783   LDI     M5310  ; 進料手臂至校正位置手動
      AND     T1000  ; 開機延遲
      INV
      FMOV    K0 D2702 K6  ; CCD>>PLCX補償   小數3位 *1000
790   LDI     M5310  ; 進料手臂至校正位置手動
      ANI     M1834  ; CCD校正機器人移動到校正點KP
      ANI     Y1025  ; 進料手臂_校正位置IN38(DI38)
      INV
      AND     M5301  ; 進料手臂允許動作
      ANI     M1842  ; CCD_校正成功(0->1)KP
      ANI     X1025  ; 進料手臂_校正位置OK(DO38)
      OUT     Y1025  ; 進料手臂_校正位置IN38(DI38)
798   LD      M5310  ; 進料手臂至校正位置手動
      AND     SM412  ; 1.0 Sec Clock
      OR      X1025  ; 進料手臂_校正位置OK(DO38)
      OUT     M5109  ; 進料手臂校正位置IN38燈
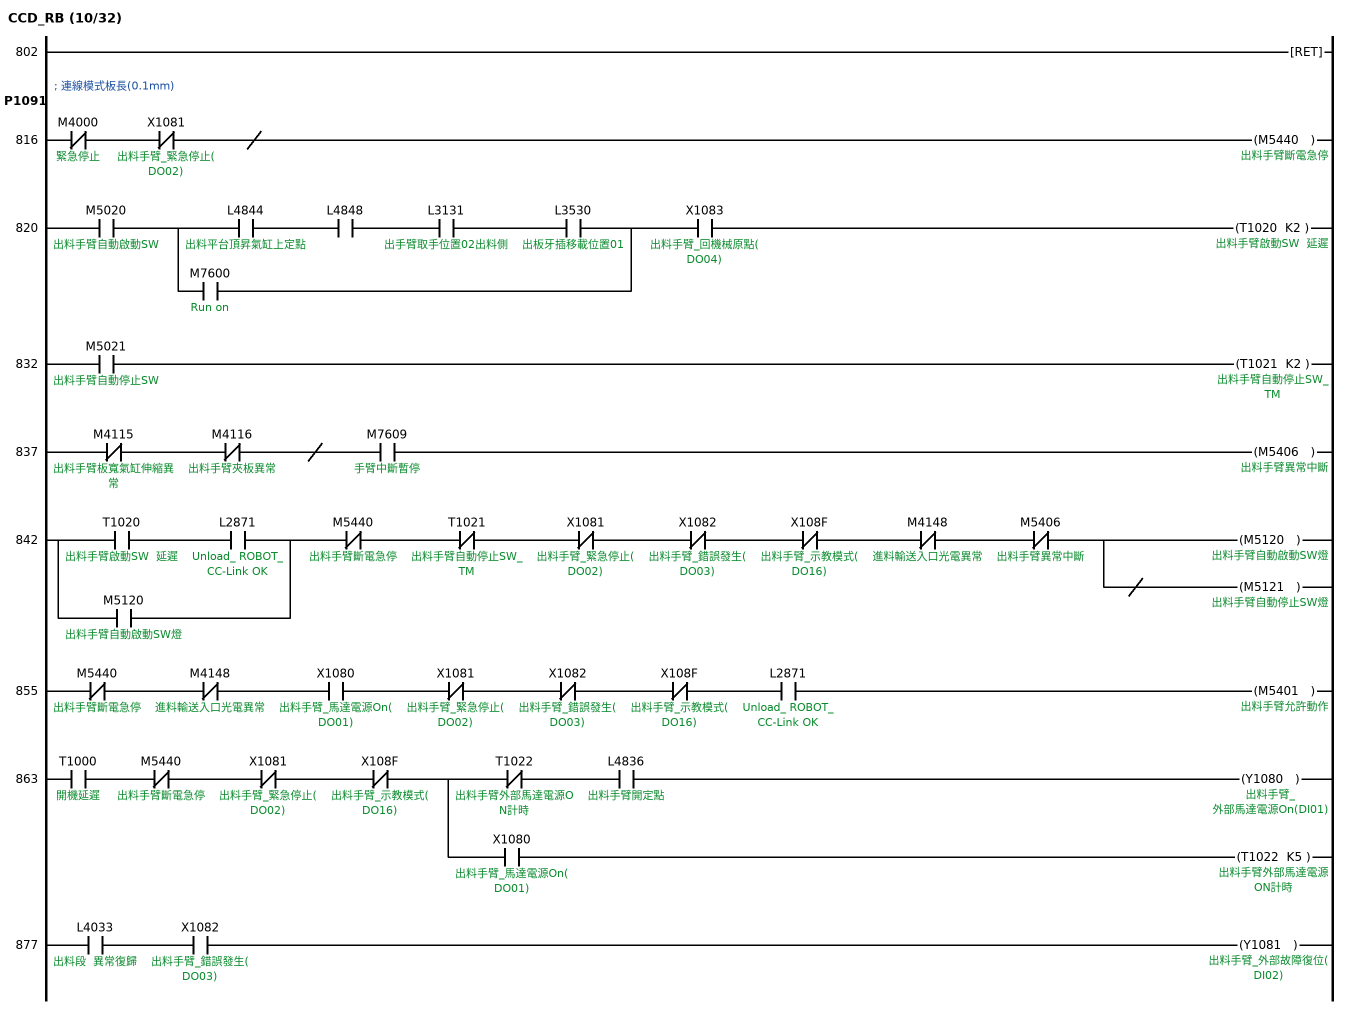
802   RET
; 連線模式板長(0.1mm)
      P1091
816   LDI     M4000  ; 緊急停止
      ANI     X1081  ; 出料手臂_緊急停止(DO02)
      INV
      OUT     M5440  ; 出料手臂斷電急停
820   LD      M5020  ; 出料手臂自動啟動SW
      LD      L4844  ; 出料平台頂昇氣缸上定點
      AND     L4848
      AND     L3131  ; 出手臂取手位置02出料側
      AND     L3530  ; 出板牙插移載位置01
      OR      M7600  ; Run on
      ANB
      AND     X1083  ; 出料手臂_回機械原點(DO04)
      OUT     T1020 K2  ; 出料手臂啟動SW  延遲
832   LD      M5021  ; 出料手臂自動停止SW
      OUT     T1021 K2  ; 出料手臂自動停止SW_TM
837   LDI     M4115  ; 出料手臂板寬氣缸伸縮異常
      ANI     M4116  ; 出料手臂夾板異常
      INV
      AND     M7609  ; 手臂中斷暫停
      OUT     M5406  ; 出料手臂異常中斷
842   LD      T1020  ; 出料手臂啟動SW  延遲
      AND     L2871  ; Unload_ ROBOT_  CC-Link OK
      OR      M5120  ; 出料手臂自動啟動SW燈
      ANI     M5440  ; 出料手臂斷電急停
      ANI     T1021  ; 出料手臂自動停止SW_TM
      ANI     X1081  ; 出料手臂_緊急停止(DO02)
      ANI     X1082  ; 出料手臂_錯誤發生(DO03)
      ANI     X108F  ; 出料手臂_示教模式(DO16)
      ANI     M4148  ; 進料輸送入口光電異常
      ANI     M5406  ; 出料手臂異常中斷
      OUT     M5120  ; 出料手臂自動啟動SW燈
      INV
      OUT     M5121  ; 出料手臂自動停止SW燈
855   LDI     M5440  ; 出料手臂斷電急停
      ANI     M4148  ; 進料輸送入口光電異常
      AND     X1080  ; 出料手臂_馬達電源On(DO01)
      ANI     X1081  ; 出料手臂_緊急停止(DO02)
      ANI     X1082  ; 出料手臂_錯誤發生(DO03)
      ANI     X108F  ; 出料手臂_示教模式(DO16)
      AND     L2871  ; Unload_ ROBOT_  CC-Link OK
      OUT     M5401  ; 出料手臂允許動作
863   LD      T1000  ; 開機延遲
      ANI     M5440  ; 出料手臂斷電急停
      ANI     X1081  ; 出料手臂_緊急停止(DO02)
      ANI     X108F  ; 出料手臂_示教模式(DO16)
      MPS
      ANI     T1022  ; 出料手臂外部馬達電源ON計時
      AND     L4836  ; 出料手臂開定點
      OUT     Y1080  ; 出料手臂_外部馬達電源On(DI01)
      MPP
      AND     X1080  ; 出料手臂_馬達電源On(DO01)
      OUT     T1022 K5  ; 出料手臂外部馬達電源ON計時
877   LD      L4033  ; 出料段  異常復歸
      AND     X1082  ; 出料手臂_錯誤發生(DO03)
      OUT     Y1081  ; 出料手臂_外部故障復位(DI02)
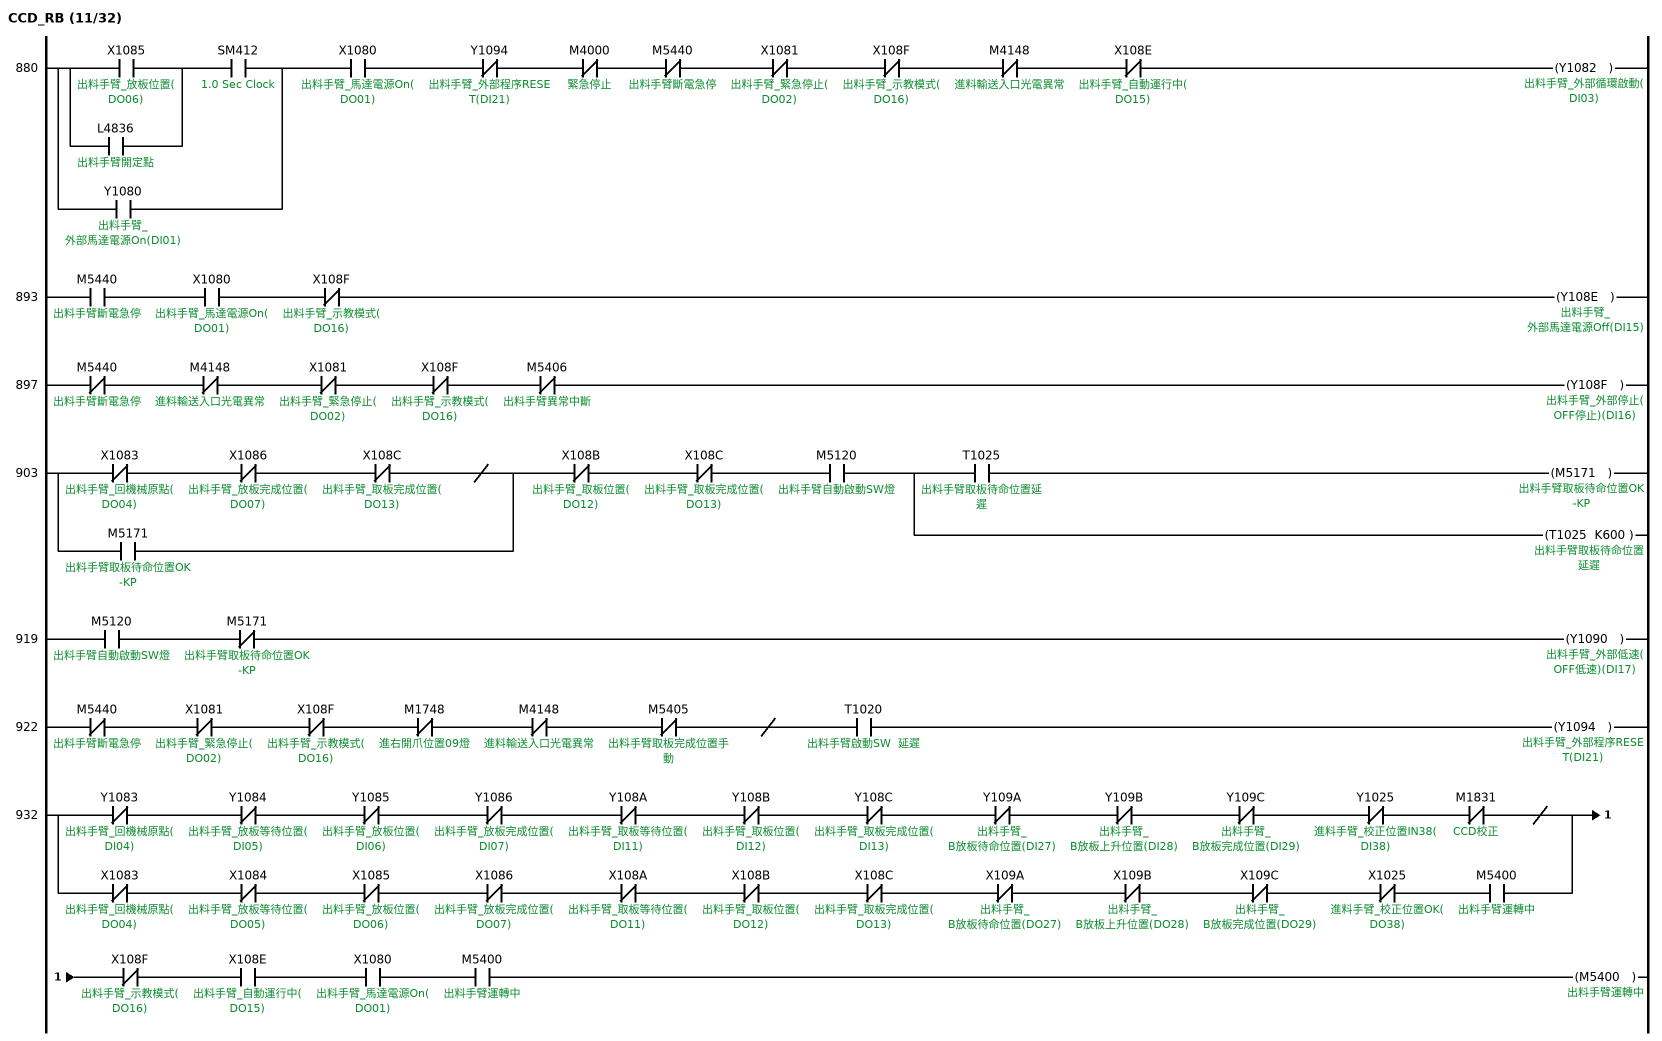
880   LD      X1085  ; 出料手臂_放板位置(DO06)
      OR      L4836  ; 出料手臂開定點
      AND     SM412  ; 1.0 Sec Clock
      OR      Y1080  ; 出料手臂_外部馬達電源On(DI01)
      AND     X1080  ; 出料手臂_馬達電源On(DO01)
      ANI     Y1094  ; 出料手臂_外部程序RESET(DI21)
      ANI     M4000  ; 緊急停止
      ANI     M5440  ; 出料手臂斷電急停
      ANI     X1081  ; 出料手臂_緊急停止(DO02)
      ANI     X108F  ; 出料手臂_示教模式(DO16)
      ANI     M4148  ; 進料輸送入口光電異常
      ANI     X108E  ; 出料手臂_自動運行中(DO15)
      OUT     Y1082  ; 出料手臂_外部循環啟動(DI03)
893   LD      M5440  ; 出料手臂斷電急停
      AND     X1080  ; 出料手臂_馬達電源On(DO01)
      ANI     X108F  ; 出料手臂_示教模式(DO16)
      OUT     Y108E  ; 出料手臂_外部馬達電源Off(DI15)
897   LDI     M5440  ; 出料手臂斷電急停
      ANI     M4148  ; 進料輸送入口光電異常
      ANI     X1081  ; 出料手臂_緊急停止(DO02)
      ANI     X108F  ; 出料手臂_示教模式(DO16)
      ANI     M5406  ; 出料手臂異常中斷
      OUT     Y108F  ; 出料手臂_外部停止(OFF停止)(DI16)
903   LDI     X1083  ; 出料手臂_回機械原點(DO04)
      ANI     X1086  ; 出料手臂_放板完成位置(DO07)
      ANI     X108C  ; 出料手臂_取板完成位置(DO13)
      INV
      OR      M5171  ; 出料手臂取板待命位置OK-KP
      ANI     X108B  ; 出料手臂_取板位置(DO12)
      ANI     X108C  ; 出料手臂_取板完成位置(DO13)
      AND     M5120  ; 出料手臂自動啟動SW燈
      MPS
      AND     T1025  ; 出料手臂取板待命位置延遲
      OUT     M5171  ; 出料手臂取板待命位置OK-KP
      MPP
      OUT     T1025 K600  ; 出料手臂取板待命位置延遲
919   LD      M5120  ; 出料手臂自動啟動SW燈
      ANI     M5171  ; 出料手臂取板待命位置OK-KP
      OUT     Y1090  ; 出料手臂_外部低速(OFF低速)(DI17)
922   LDI     M5440  ; 出料手臂斷電急停
      ANI     X1081  ; 出料手臂_緊急停止(DO02)
      ANI     X108F  ; 出料手臂_示教模式(DO16)
      ANI     M1748  ; 進右開爪位置09燈
      ANI     M4148  ; 進料輸送入口光電異常
      ANI     M5405  ; 出料手臂取板完成位置手動
      INV
      AND     T1020  ; 出料手臂啟動SW  延遲
      OUT     Y1094  ; 出料手臂_外部程序RESET(DI21)
932   LDI     Y1083  ; 出料手臂_回機械原點(DI04)
      ANI     Y1084  ; 出料手臂_放板等待位置(DI05)
      ANI     Y1085  ; 出料手臂_放板位置(DI06)
      ANI     Y1086  ; 出料手臂_放板完成位置(DI07)
      ANI     Y108A  ; 出料手臂_取板等待位置(DI11)
      ANI     Y108B  ; 出料手臂_取板位置(DI12)
      ANI     Y108C  ; 出料手臂_取板完成位置(DI13)
      ANI     Y109A  ; 出料手臂_B放板待命位置(DI27)
      ANI     Y109B  ; 出料手臂_B放板上升位置(DI28)
      ANI     Y109C  ; 出料手臂_B放板完成位置(DI29)
      ANI     Y1025  ; 進料手臂_校正位置IN38(DI38)
      ANI     M1831  ; CCD校正
      INV
      LDI     X1083  ; 出料手臂_回機械原點(DO04)
      ANI     X1084  ; 出料手臂_放板等待位置(DO05)
      ANI     X1085  ; 出料手臂_放板位置(DO06)
      ANI     X1086  ; 出料手臂_放板完成位置(DO07)
      ANI     X108A  ; 出料手臂_取板等待位置(DO11)
      ANI     X108B  ; 出料手臂_取板位置(DO12)
      ANI     X108C  ; 出料手臂_取板完成位置(DO13)
      ANI     X109A  ; 出料手臂_B放板待命位置(DO27)
      ANI     X109B  ; 出料手臂_B放板上升位置(DO28)
      ANI     X109C  ; 出料手臂_B放板完成位置(DO29)
      ANI     X1025  ; 進料手臂_校正位置OK(DO38)
      AND     M5400  ; 出料手臂運轉中
      ORB
      ANI     X108F  ; 出料手臂_示教模式(DO16)
      AND     X108E  ; 出料手臂_自動運行中(DO15)
      AND     X1080  ; 出料手臂_馬達電源On(DO01)
      AND     M5400  ; 出料手臂運轉中
      OUT     M5400  ; 出料手臂運轉中
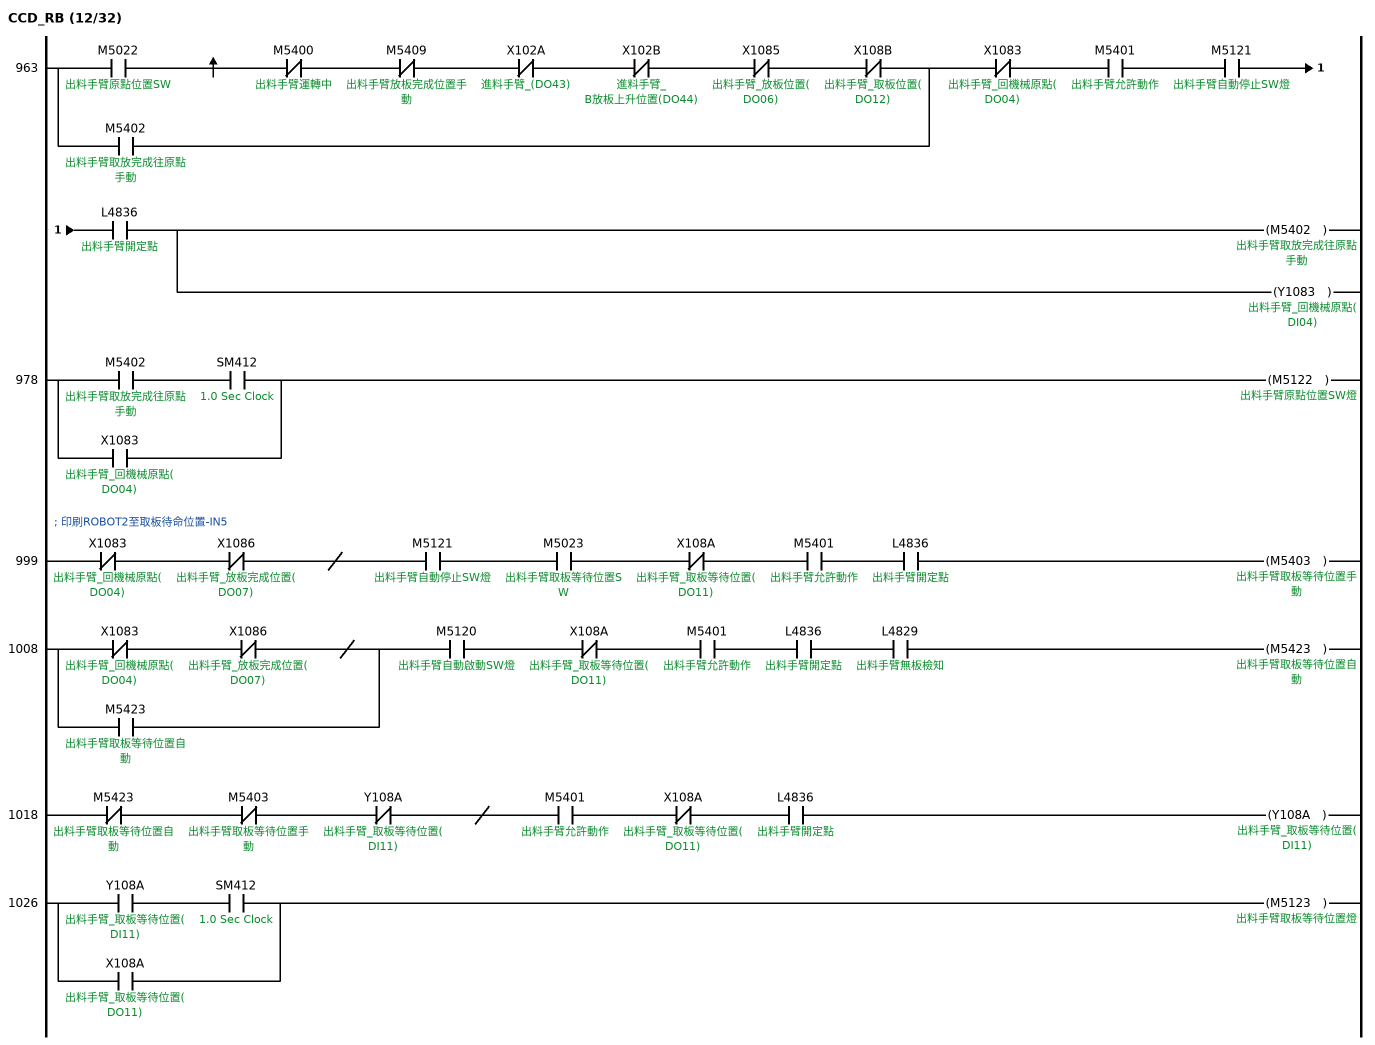
963   LD      M5022  ; 出料手臂原點位置SW
      MEP
      ANI     M5400  ; 出料手臂運轉中
      ANI     M5409  ; 出料手臂放板完成位置手動
      ANI     X102A  ; 進料手臂_(DO43)
      ANI     X102B  ; 進料手臂_B放板上升位置(DO44)
      ANI     X1085  ; 出料手臂_放板位置(DO06)
      ANI     X108B  ; 出料手臂_取板位置(DO12)
      OR      M5402  ; 出料手臂取放完成往原點手動
      ANI     X1083  ; 出料手臂_回機械原點(DO04)
      AND     M5401  ; 出料手臂允許動作
      AND     M5121  ; 出料手臂自動停止SW燈
      AND     L4836  ; 出料手臂開定點
      OUT     M5402  ; 出料手臂取放完成往原點手動
      OUT     Y1083  ; 出料手臂_回機械原點(DI04)
978   LD      M5402  ; 出料手臂取放完成往原點手動
      AND     SM412  ; 1.0 Sec Clock
      OR      X1083  ; 出料手臂_回機械原點(DO04)
      OUT     M5122  ; 出料手臂原點位置SW燈
; 印刷ROBOT2至取板待命位置-IN5
999   LDI     X1083  ; 出料手臂_回機械原點(DO04)
      ANI     X1086  ; 出料手臂_放板完成位置(DO07)
      INV
      AND     M5121  ; 出料手臂自動停止SW燈
      AND     M5023  ; 出料手臂取板等待位置SW
      ANI     X108A  ; 出料手臂_取板等待位置(DO11)
      AND     M5401  ; 出料手臂允許動作
      AND     L4836  ; 出料手臂開定點
      OUT     M5403  ; 出料手臂取板等待位置手動
1008  LDI     X1083  ; 出料手臂_回機械原點(DO04)
      ANI     X1086  ; 出料手臂_放板完成位置(DO07)
      INV
      OR      M5423  ; 出料手臂取板等待位置自動
      AND     M5120  ; 出料手臂自動啟動SW燈
      ANI     X108A  ; 出料手臂_取板等待位置(DO11)
      AND     M5401  ; 出料手臂允許動作
      AND     L4836  ; 出料手臂開定點
      AND     L4829  ; 出料手臂無板檢知
      OUT     M5423  ; 出料手臂取板等待位置自動
1018  LDI     M5423  ; 出料手臂取板等待位置自動
      ANI     M5403  ; 出料手臂取板等待位置手動
      ANI     Y108A  ; 出料手臂_取板等待位置(DI11)
      INV
      AND     M5401  ; 出料手臂允許動作
      ANI     X108A  ; 出料手臂_取板等待位置(DO11)
      AND     L4836  ; 出料手臂開定點
      OUT     Y108A  ; 出料手臂_取板等待位置(DI11)
1026  LD      Y108A  ; 出料手臂_取板等待位置(DI11)
      AND     SM412  ; 1.0 Sec Clock
      OR      X108A  ; 出料手臂_取板等待位置(DO11)
      OUT     M5123  ; 出料手臂取板等待位置燈
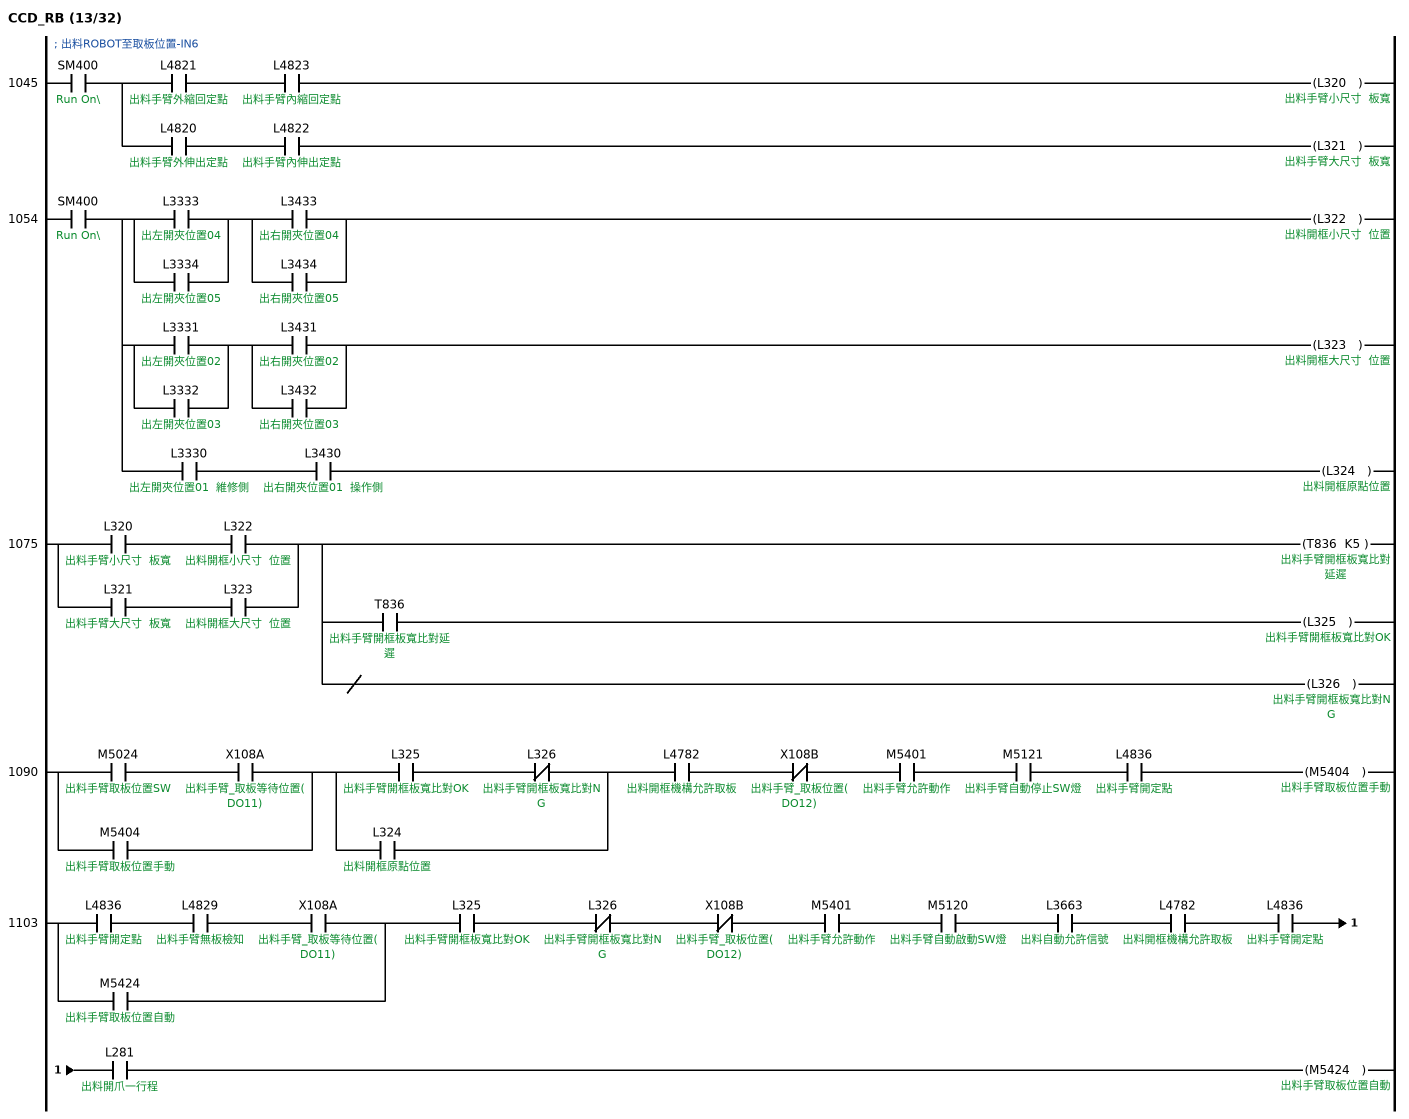
; 出料ROBOT至取板位置-IN6
1045  LD      SM400  ; Run On\
      MPS
      AND     L4821  ; 出料手臂外縮回定點
      AND     L4823  ; 出料手臂內縮回定點
      OUT     L320  ; 出料手臂小尺寸  板寬
      MPP
      AND     L4820  ; 出料手臂外伸出定點
      AND     L4822  ; 出料手臂內伸出定點
      OUT     L321  ; 出料手臂大尺寸  板寬
1054  LD      SM400  ; Run On\
      MPS
      LD      L3333  ; 出左開夾位置04
      OR      L3334  ; 出左開夾位置05
      ANB
      LD      L3433  ; 出右開夾位置04
      OR      L3434  ; 出右開夾位置05
      ANB
      OUT     L322  ; 出料開框小尺寸  位置
      MRD
      LD      L3331  ; 出左開夾位置02
      OR      L3332  ; 出左開夾位置03
      ANB
      LD      L3431  ; 出右開夾位置02
      OR      L3432  ; 出右開夾位置03
      ANB
      OUT     L323  ; 出料開框大尺寸  位置
      MPP
      AND     L3330  ; 出左開夾位置01  維修側
      AND     L3430  ; 出右開夾位置01  操作側
      OUT     L324  ; 出料開框原點位置
1075  LD      L320  ; 出料手臂小尺寸  板寬
      AND     L322  ; 出料開框小尺寸  位置
      LD      L321  ; 出料手臂大尺寸  板寬
      AND     L323  ; 出料開框大尺寸  位置
      ORB
      OUT     T836 K5  ; 出料手臂開框板寬比對延遲
      MPS
      AND     T836  ; 出料手臂開框板寬比對延遲
      OUT     L325  ; 出料手臂開框板寬比對OK
      MPP
      INV
      OUT     L326  ; 出料手臂開框板寬比對NG
1090  LD      M5024  ; 出料手臂取板位置SW
      AND     X108A  ; 出料手臂_取板等待位置(DO11)
      OR      M5404  ; 出料手臂取板位置手動
      LD      L325  ; 出料手臂開框板寬比對OK
      ANI     L326  ; 出料手臂開框板寬比對NG
      OR      L324  ; 出料開框原點位置
      ANB
      AND     L4782  ; 出料開框機構允許取板
      ANI     X108B  ; 出料手臂_取板位置(DO12)
      AND     M5401  ; 出料手臂允許動作
      AND     M5121  ; 出料手臂自動停止SW燈
      AND     L4836  ; 出料手臂開定點
      OUT     M5404  ; 出料手臂取板位置手動
1103  LD      L4836  ; 出料手臂開定點
      AND     L4829  ; 出料手臂無板檢知
      AND     X108A  ; 出料手臂_取板等待位置(DO11)
      OR      M5424  ; 出料手臂取板位置自動
      AND     L325  ; 出料手臂開框板寬比對OK
      ANI     L326  ; 出料手臂開框板寬比對NG
      ANI     X108B  ; 出料手臂_取板位置(DO12)
      AND     M5401  ; 出料手臂允許動作
      AND     M5120  ; 出料手臂自動啟動SW燈
      AND     L3663  ; 出料自動允許信號
      AND     L4782  ; 出料開框機構允許取板
      AND     L4836  ; 出料手臂開定點
      AND     L281  ; 出料開爪一行程
      OUT     M5424  ; 出料手臂取板位置自動
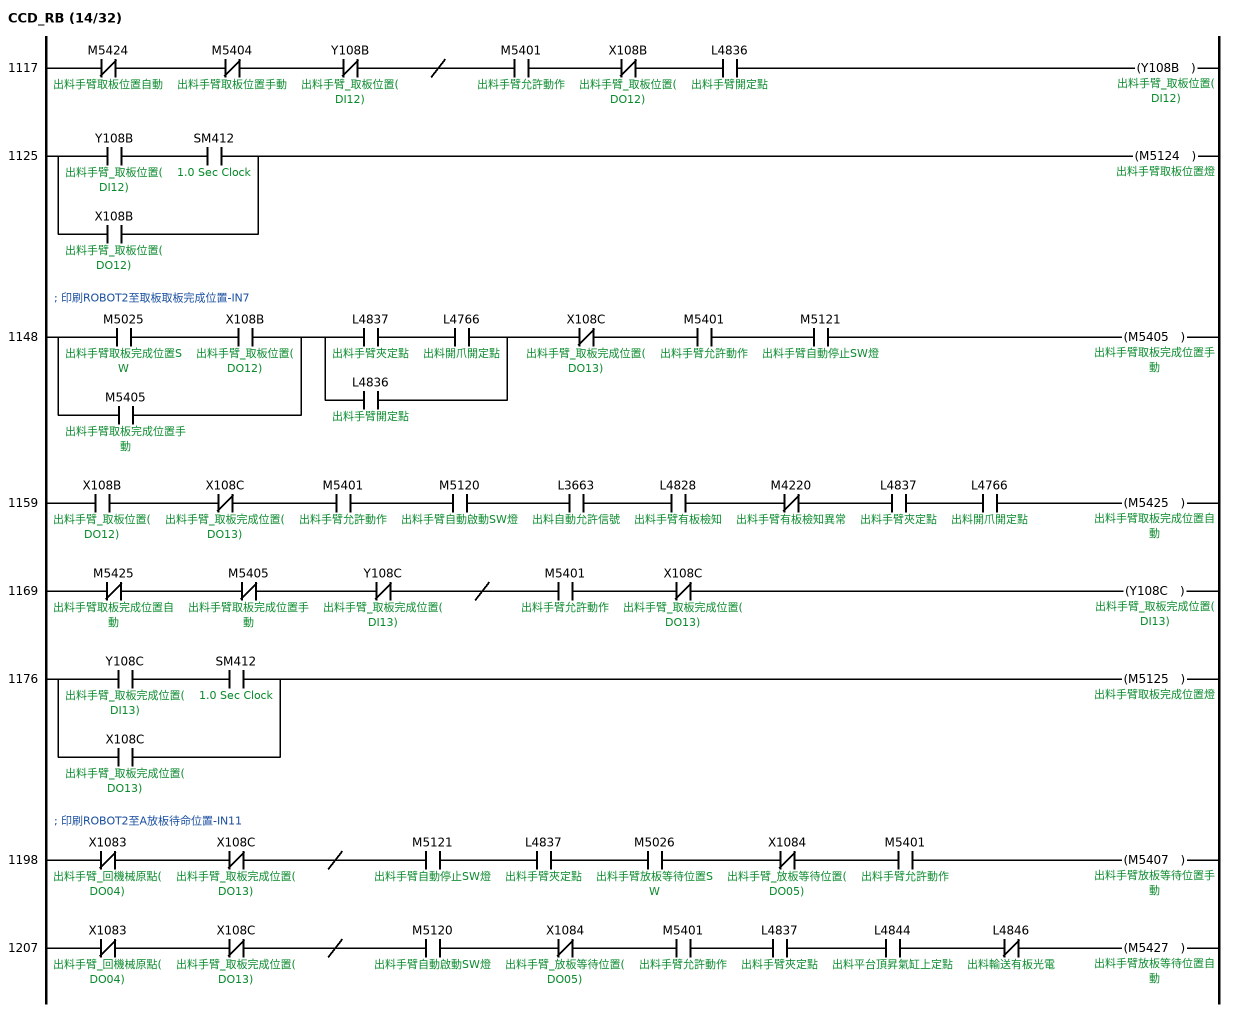
1117  LDI     M5424  ; 出料手臂取板位置自動
      ANI     M5404  ; 出料手臂取板位置手動
      ANI     Y108B  ; 出料手臂_取板位置(DI12)
      INV
      AND     M5401  ; 出料手臂允許動作
      ANI     X108B  ; 出料手臂_取板位置(DO12)
      AND     L4836  ; 出料手臂開定點
      OUT     Y108B  ; 出料手臂_取板位置(DI12)
1125  LD      Y108B  ; 出料手臂_取板位置(DI12)
      AND     SM412  ; 1.0 Sec Clock
      OR      X108B  ; 出料手臂_取板位置(DO12)
      OUT     M5124  ; 出料手臂取板位置燈
; 印刷ROBOT2至取板取板完成位置-IN7
1148  LD      M5025  ; 出料手臂取板完成位置SW
      AND     X108B  ; 出料手臂_取板位置(DO12)
      OR      M5405  ; 出料手臂取板完成位置手動
      LD      L4837  ; 出料手臂夾定點
      AND     L4766  ; 出料開爪開定點
      OR      L4836  ; 出料手臂開定點
      ANB
      ANI     X108C  ; 出料手臂_取板完成位置(DO13)
      AND     M5401  ; 出料手臂允許動作
      AND     M5121  ; 出料手臂自動停止SW燈
      OUT     M5405  ; 出料手臂取板完成位置手動
1159  LD      X108B  ; 出料手臂_取板位置(DO12)
      ANI     X108C  ; 出料手臂_取板完成位置(DO13)
      AND     M5401  ; 出料手臂允許動作
      AND     M5120  ; 出料手臂自動啟動SW燈
      AND     L3663  ; 出料自動允許信號
      AND     L4828  ; 出料手臂有板檢知
      ANI     M4220  ; 出料手臂有板檢知異常
      AND     L4837  ; 出料手臂夾定點
      AND     L4766  ; 出料開爪開定點
      OUT     M5425  ; 出料手臂取板完成位置自動
1169  LDI     M5425  ; 出料手臂取板完成位置自動
      ANI     M5405  ; 出料手臂取板完成位置手動
      ANI     Y108C  ; 出料手臂_取板完成位置(DI13)
      INV
      AND     M5401  ; 出料手臂允許動作
      ANI     X108C  ; 出料手臂_取板完成位置(DO13)
      OUT     Y108C  ; 出料手臂_取板完成位置(DI13)
1176  LD      Y108C  ; 出料手臂_取板完成位置(DI13)
      AND     SM412  ; 1.0 Sec Clock
      OR      X108C  ; 出料手臂_取板完成位置(DO13)
      OUT     M5125  ; 出料手臂取板完成位置燈
; 印刷ROBOT2至A放板待命位置-IN11
1198  LDI     X1083  ; 出料手臂_回機械原點(DO04)
      ANI     X108C  ; 出料手臂_取板完成位置(DO13)
      INV
      AND     M5121  ; 出料手臂自動停止SW燈
      AND     L4837  ; 出料手臂夾定點
      AND     M5026  ; 出料手臂放板等待位置SW
      ANI     X1084  ; 出料手臂_放板等待位置(DO05)
      AND     M5401  ; 出料手臂允許動作
      OUT     M5407  ; 出料手臂放板等待位置手動
1207  LDI     X1083  ; 出料手臂_回機械原點(DO04)
      ANI     X108C  ; 出料手臂_取板完成位置(DO13)
      INV
      AND     M5120  ; 出料手臂自動啟動SW燈
      ANI     X1084  ; 出料手臂_放板等待位置(DO05)
      AND     M5401  ; 出料手臂允許動作
      AND     L4837  ; 出料手臂夾定點
      AND     L4844  ; 出料平台頂昇氣缸上定點
      ANI     L4846  ; 出料輸送有板光電
      OUT     M5427  ; 出料手臂放板等待位置自動
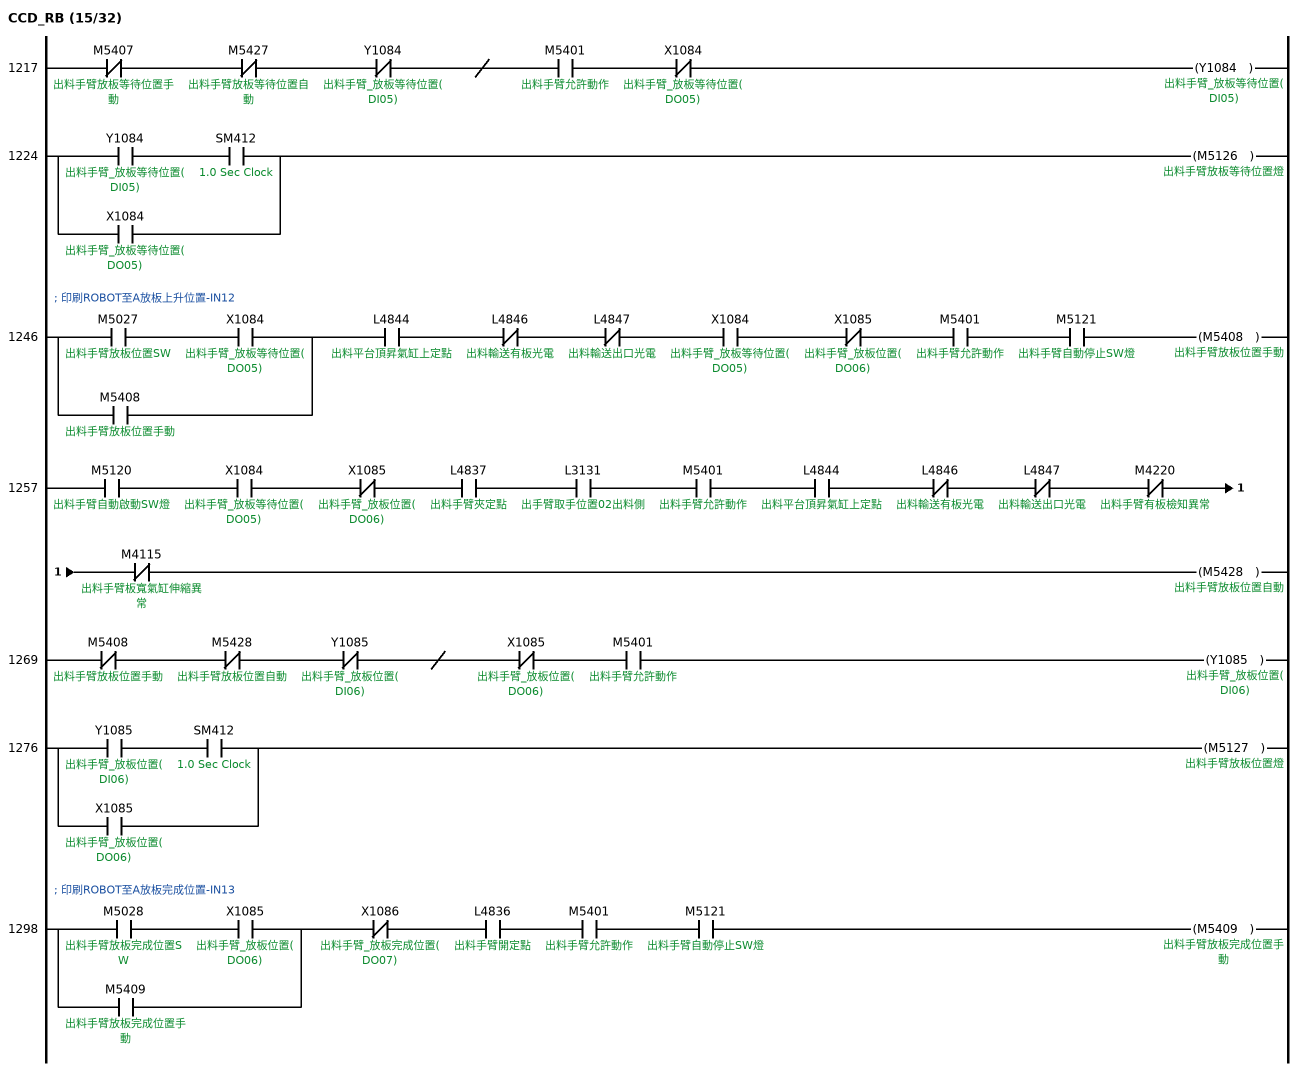
1217  LDI     M5407  ; 出料手臂放板等待位置手動
      ANI     M5427  ; 出料手臂放板等待位置自動
      ANI     Y1084  ; 出料手臂_放板等待位置(DI05)
      INV
      AND     M5401  ; 出料手臂允許動作
      ANI     X1084  ; 出料手臂_放板等待位置(DO05)
      OUT     Y1084  ; 出料手臂_放板等待位置(DI05)
1224  LD      Y1084  ; 出料手臂_放板等待位置(DI05)
      AND     SM412  ; 1.0 Sec Clock
      OR      X1084  ; 出料手臂_放板等待位置(DO05)
      OUT     M5126  ; 出料手臂放板等待位置燈
; 印刷ROBOT至A放板上升位置-IN12
1246  LD      M5027  ; 出料手臂放板位置SW
      AND     X1084  ; 出料手臂_放板等待位置(DO05)
      OR      M5408  ; 出料手臂放板位置手動
      AND     L4844  ; 出料平台頂昇氣缸上定點
      ANI     L4846  ; 出料輸送有板光電
      ANI     L4847  ; 出料輸送出口光電
      AND     X1084  ; 出料手臂_放板等待位置(DO05)
      ANI     X1085  ; 出料手臂_放板位置(DO06)
      AND     M5401  ; 出料手臂允許動作
      AND     M5121  ; 出料手臂自動停止SW燈
      OUT     M5408  ; 出料手臂放板位置手動
1257  LD      M5120  ; 出料手臂自動啟動SW燈
      AND     X1084  ; 出料手臂_放板等待位置(DO05)
      ANI     X1085  ; 出料手臂_放板位置(DO06)
      AND     L4837  ; 出料手臂夾定點
      AND     L3131  ; 出手臂取手位置02出料側
      AND     M5401  ; 出料手臂允許動作
      AND     L4844  ; 出料平台頂昇氣缸上定點
      ANI     L4846  ; 出料輸送有板光電
      ANI     L4847  ; 出料輸送出口光電
      ANI     M4220  ; 出料手臂有板檢知異常
      ANI     M4115  ; 出料手臂板寬氣缸伸縮異常
      OUT     M5428  ; 出料手臂放板位置自動
1269  LDI     M5408  ; 出料手臂放板位置手動
      ANI     M5428  ; 出料手臂放板位置自動
      ANI     Y1085  ; 出料手臂_放板位置(DI06)
      INV
      ANI     X1085  ; 出料手臂_放板位置(DO06)
      AND     M5401  ; 出料手臂允許動作
      OUT     Y1085  ; 出料手臂_放板位置(DI06)
1276  LD      Y1085  ; 出料手臂_放板位置(DI06)
      AND     SM412  ; 1.0 Sec Clock
      OR      X1085  ; 出料手臂_放板位置(DO06)
      OUT     M5127  ; 出料手臂放板位置燈
; 印刷ROBOT至A放板完成位置-IN13
1298  LD      M5028  ; 出料手臂放板完成位置SW
      AND     X1085  ; 出料手臂_放板位置(DO06)
      OR      M5409  ; 出料手臂放板完成位置手動
      ANI     X1086  ; 出料手臂_放板完成位置(DO07)
      AND     L4836  ; 出料手臂開定點
      AND     M5401  ; 出料手臂允許動作
      AND     M5121  ; 出料手臂自動停止SW燈
      OUT     M5409  ; 出料手臂放板完成位置手動
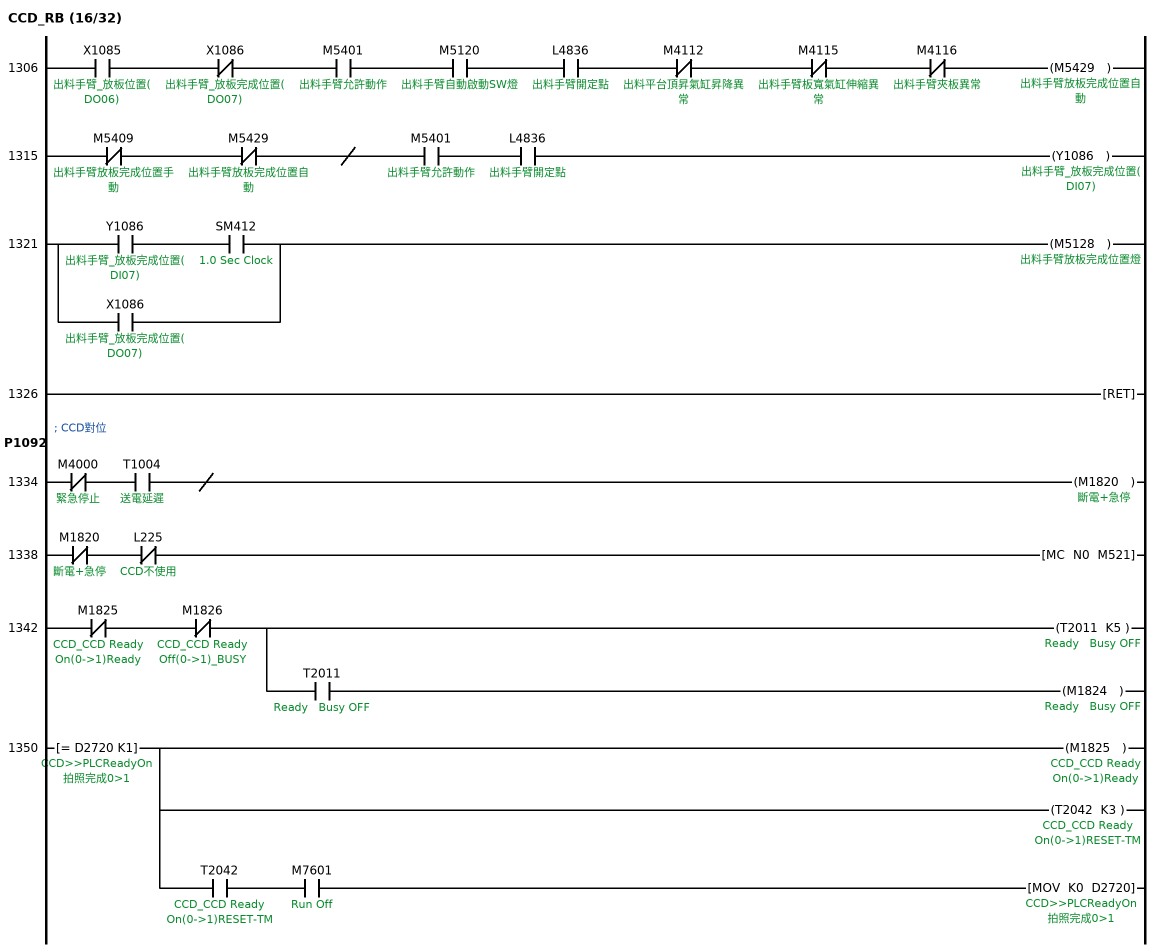
1306  LD      X1085  ; 出料手臂_放板位置(DO06)
      ANI     X1086  ; 出料手臂_放板完成位置(DO07)
      AND     M5401  ; 出料手臂允許動作
      AND     M5120  ; 出料手臂自動啟動SW燈
      AND     L4836  ; 出料手臂開定點
      ANI     M4112  ; 出料平台頂昇氣缸昇降異常
      ANI     M4115  ; 出料手臂板寬氣缸伸縮異常
      ANI     M4116  ; 出料手臂夾板異常
      OUT     M5429  ; 出料手臂放板完成位置自動
1315  LDI     M5409  ; 出料手臂放板完成位置手動
      ANI     M5429  ; 出料手臂放板完成位置自動
      INV
      AND     M5401  ; 出料手臂允許動作
      AND     L4836  ; 出料手臂開定點
      OUT     Y1086  ; 出料手臂_放板完成位置(DI07)
1321  LD      Y1086  ; 出料手臂_放板完成位置(DI07)
      AND     SM412  ; 1.0 Sec Clock
      OR      X1086  ; 出料手臂_放板完成位置(DO07)
      OUT     M5128  ; 出料手臂放板完成位置燈
1326  RET
; CCD對位
      P1092
1334  LDI     M4000  ; 緊急停止
      AND     T1004  ; 送電延遲
      INV
      OUT     M1820  ; 斷電+急停
1338  LDI     M1820  ; 斷電+急停
      ANI     L225  ; CCD不使用
      MC      N0 M521
1342  LDI     M1825  ; CCD_CCD Ready On(0->1)Ready
      ANI     M1826  ; CCD_CCD Ready Off(0->1)_BUSY
      OUT     T2011 K5  ; Ready   Busy OFF
      AND     T2011  ; Ready   Busy OFF
      OUT     M1824  ; Ready   Busy OFF
1350  LD=     D2720 K1  ; CCD>>PLCReadyOn 拍照完成0>1
      OUT     M1825  ; CCD_CCD Ready On(0->1)Ready
      OUT     T2042 K3  ; CCD_CCD Ready On(0->1)RESET-TM
      AND     T2042  ; CCD_CCD Ready On(0->1)RESET-TM
      AND     M7601  ; Run Off
      MOV     K0 D2720
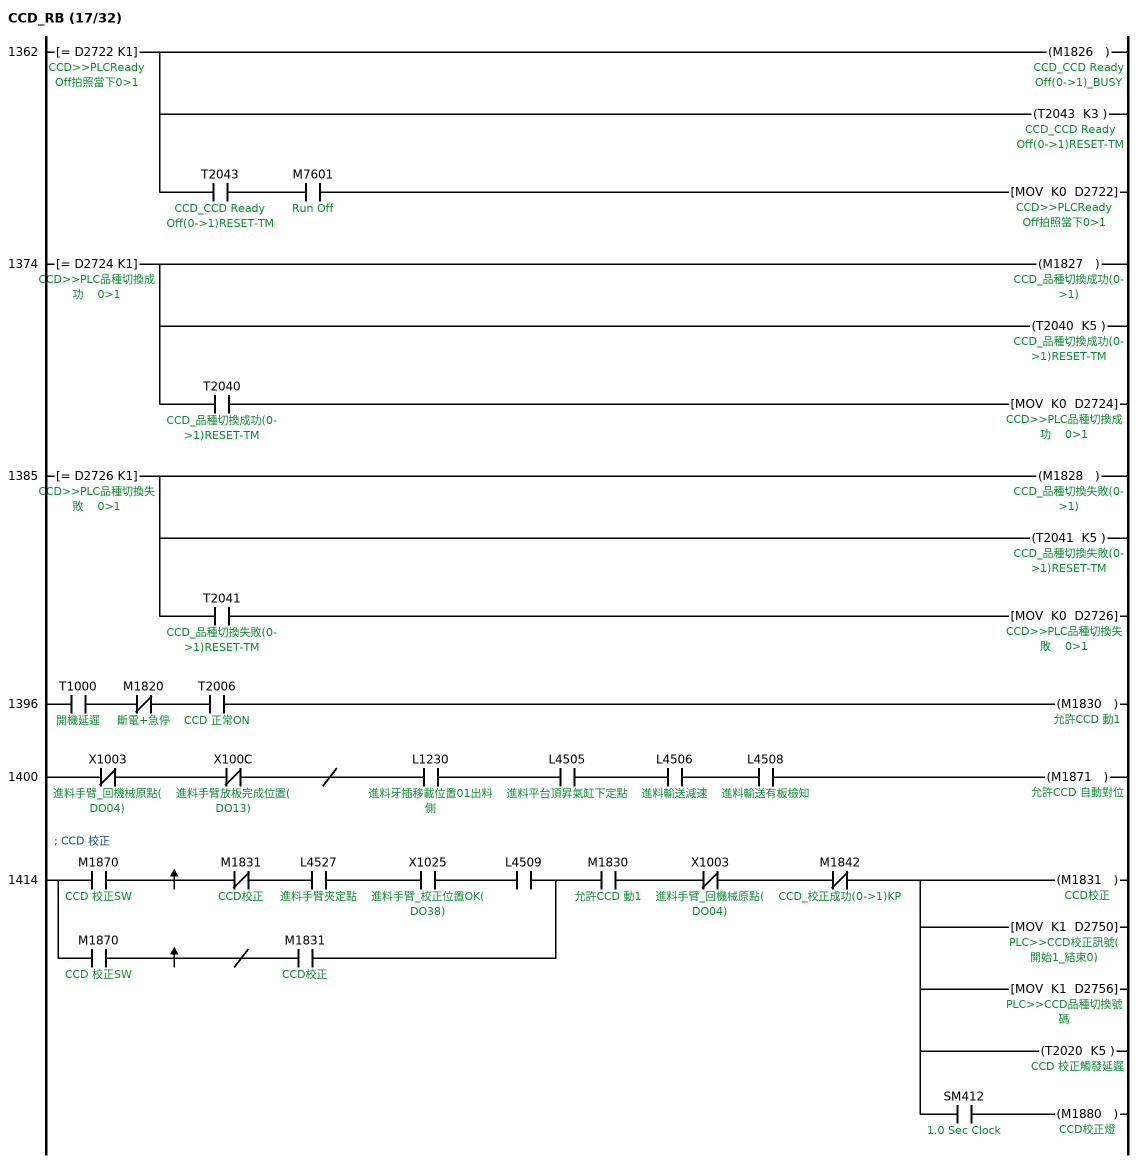
1362  LD=     D2722 K1  ; CCD>>PLCReadyOff拍照當下0>1
      OUT     M1826  ; CCD_CCD Ready Off(0->1)_BUSY
      OUT     T2043 K3  ; CCD_CCD Ready Off(0->1)RESET-TM
      AND     T2043  ; CCD_CCD Ready Off(0->1)RESET-TM
      AND     M7601  ; Run Off
      MOV     K0 D2722
1374  LD=     D2724 K1  ; CCD>>PLC品種切換成功    0>1
      OUT     M1827  ; CCD_品種切換成功(0->1)
      OUT     T2040 K5  ; CCD_品種切換成功(0->1)RESET-TM
      AND     T2040  ; CCD_品種切換成功(0->1)RESET-TM
      MOV     K0 D2724
1385  LD=     D2726 K1  ; CCD>>PLC品種切換失敗    0>1
      OUT     M1828  ; CCD_品種切換失敗(0->1)
      OUT     T2041 K5  ; CCD_品種切換失敗(0->1)RESET-TM
      AND     T2041  ; CCD_品種切換失敗(0->1)RESET-TM
      MOV     K0 D2726
1396  LD      T1000  ; 開機延遲
      ANI     M1820  ; 斷電+急停
      AND     T2006  ; CCD 正常ON
      OUT     M1830  ; 允許CCD 動1
1400  LDI     X1003  ; 進料手臂_回機械原點(DO04)
      ANI     X100C  ; 進料手臂放板完成位置(DO13)
      INV
      AND     L1230  ; 進料牙插移載位置01出料側
      AND     L4505  ; 進料平台頂昇氣缸下定點
      AND     L4506  ; 進料輸送減速
      AND     L4508  ; 進料輸送有板檢知
      OUT     M1871  ; 允許CCD 自動對位
; CCD 校正
1414  LD      M1870  ; CCD 校正SW
      MEP
      ANI     M1831  ; CCD校正
      AND     L4527  ; 進料手臂夾定點
      AND     X1025  ; 進料手臂_校正位置OK(DO38)
      AND     L4509
      LD      M1870  ; CCD 校正SW
      MEP
      INV
      AND     M1831  ; CCD校正
      ORB
      AND     M1830  ; 允許CCD 動1
      ANI     X1003  ; 進料手臂_回機械原點(DO04)
      ANI     M1842  ; CCD_校正成功(0->1)KP
      OUT     M1831  ; CCD校正
      MOV     K1 D2750  ; PLC>>CCD校正訊號(開始1_結束0)
      MOV     K1 D2756  ; PLC>>CCD品種切換號碼
      OUT     T2020 K5  ; CCD 校正觸發延遲
      AND     SM412  ; 1.0 Sec Clock
      OUT     M1880  ; CCD校正燈
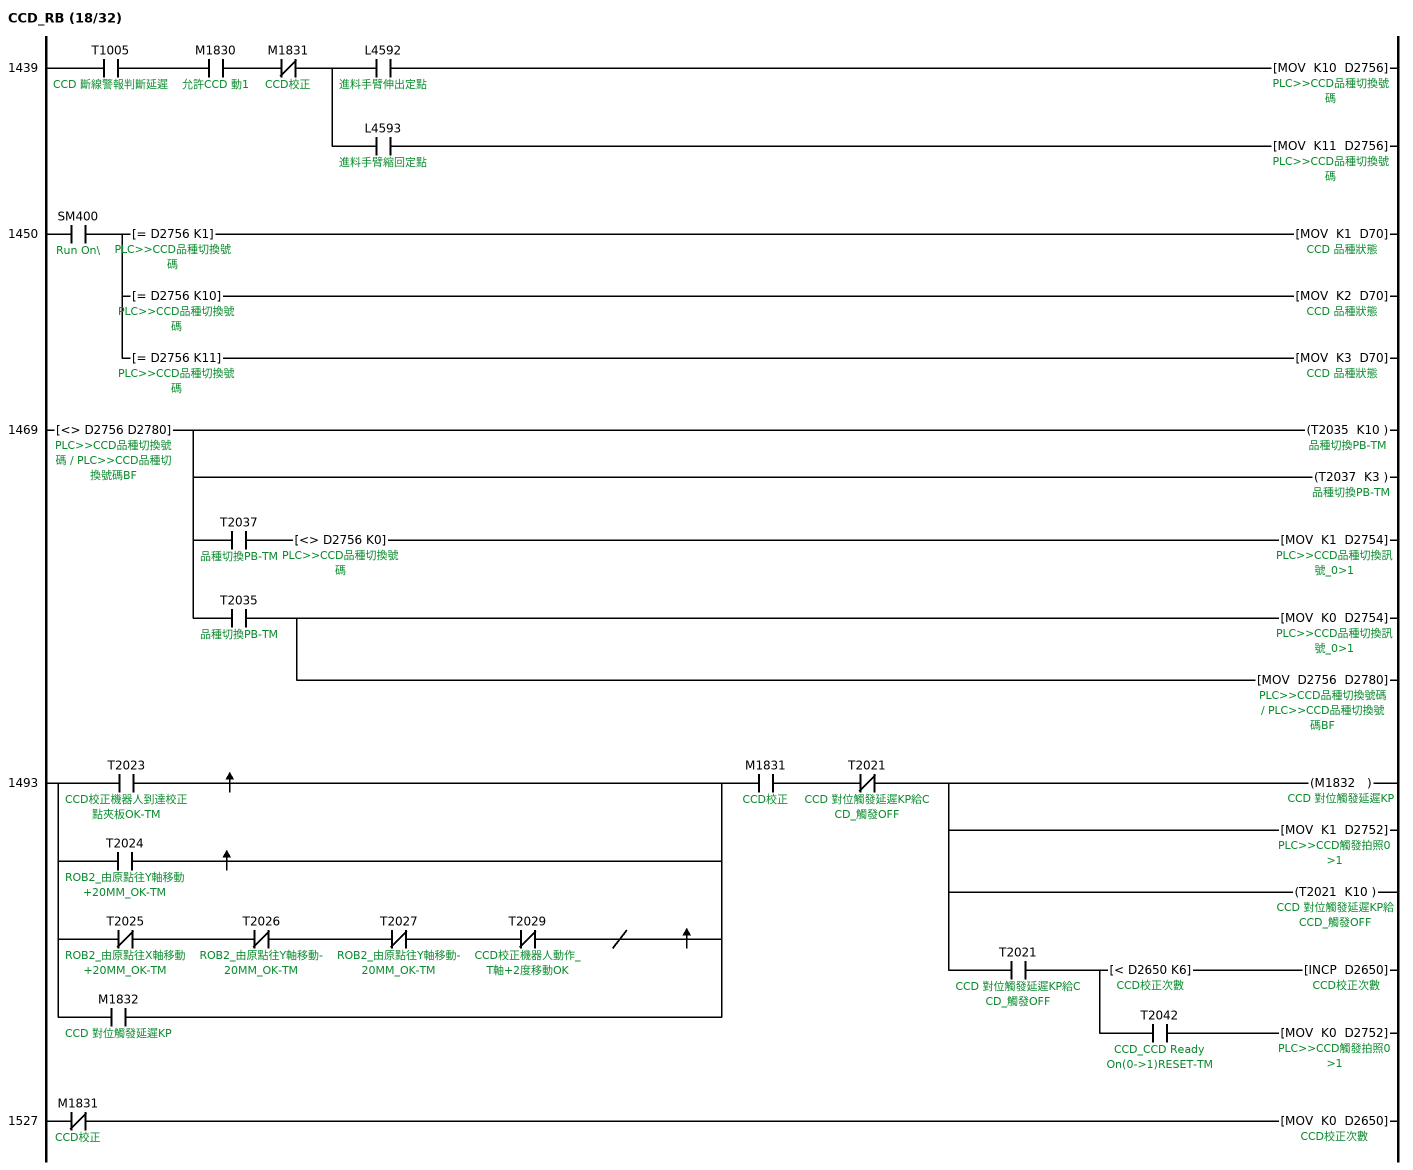
1439  LD      T1005  ; CCD 斷線警報判斷延遲
      AND     M1830  ; 允許CCD 動1
      ANI     M1831  ; CCD校正
      MPS
      AND     L4592  ; 進料手臂伸出定點
      MOV     K10 D2756
      MPP
      AND     L4593  ; 進料手臂縮回定點
      MOV     K11 D2756
1450  LD      SM400  ; Run On\
      MPS
      AND=    D2756 K1  ; PLC>>CCD品種切換號碼
      MOV     K1 D70  ; CCD 品種狀態
      MRD
      AND=    D2756 K10  ; PLC>>CCD品種切換號碼
      MOV     K2 D70
      MPP
      AND=    D2756 K11  ; PLC>>CCD品種切換號碼
      MOV     K3 D70
1469  LD<>    D2756 D2780  ; PLC>>CCD品種切換號碼 / PLC>>CCD品種切換號碼BF
      OUT     T2035 K10  ; 品種切換PB-TM
      OUT     T2037 K3  ; 品種切換PB-TM
      MPS
      AND     T2037  ; 品種切換PB-TM
      AND<>   D2756 K0  ; PLC>>CCD品種切換號碼
      MOV     K1 D2754  ; PLC>>CCD品種切換訊號_0>1
      MPP
      AND     T2035  ; 品種切換PB-TM
      MOV     K0 D2754
      MOV     D2756 D2780
1493  LD      T2023  ; CCD校正機器人到達校正點夾板OK-TM
      MEP
      LD      T2024  ; ROB2_由原點往Y軸移動+20MM_OK-TM
      MEP
      ORB
      LDI     T2025  ; ROB2_由原點往X軸移動+20MM_OK-TM
      ANI     T2026  ; ROB2_由原點往Y軸移動-20MM_OK-TM
      ANI     T2027  ; ROB2_由原點往Y軸移動-20MM_OK-TM
      ANI     T2029  ; CCD校正機器人動作_T軸+2度移動OK
      INV
      MEP
      ORB
      OR      M1832  ; CCD 對位觸發延遲KP
      AND     M1831  ; CCD校正
      ANI     T2021  ; CCD 對位觸發延遲KP給CCD_觸發OFF
      OUT     M1832  ; CCD 對位觸發延遲KP
      MOV     K1 D2752  ; PLC>>CCD觸發拍照0>1
      OUT     T2021 K10  ; CCD 對位觸發延遲KP給CCD_觸發OFF
      AND     T2021  ; CCD 對位觸發延遲KP給CCD_觸發OFF
      MPS
      AND<    D2650 K6  ; CCD校正次數
      INCP    D2650
      MPP
      AND     T2042  ; CCD_CCD Ready On(0->1)RESET-TM
      MOV     K0 D2752
1527  LDI     M1831  ; CCD校正
      MOV     K0 D2650
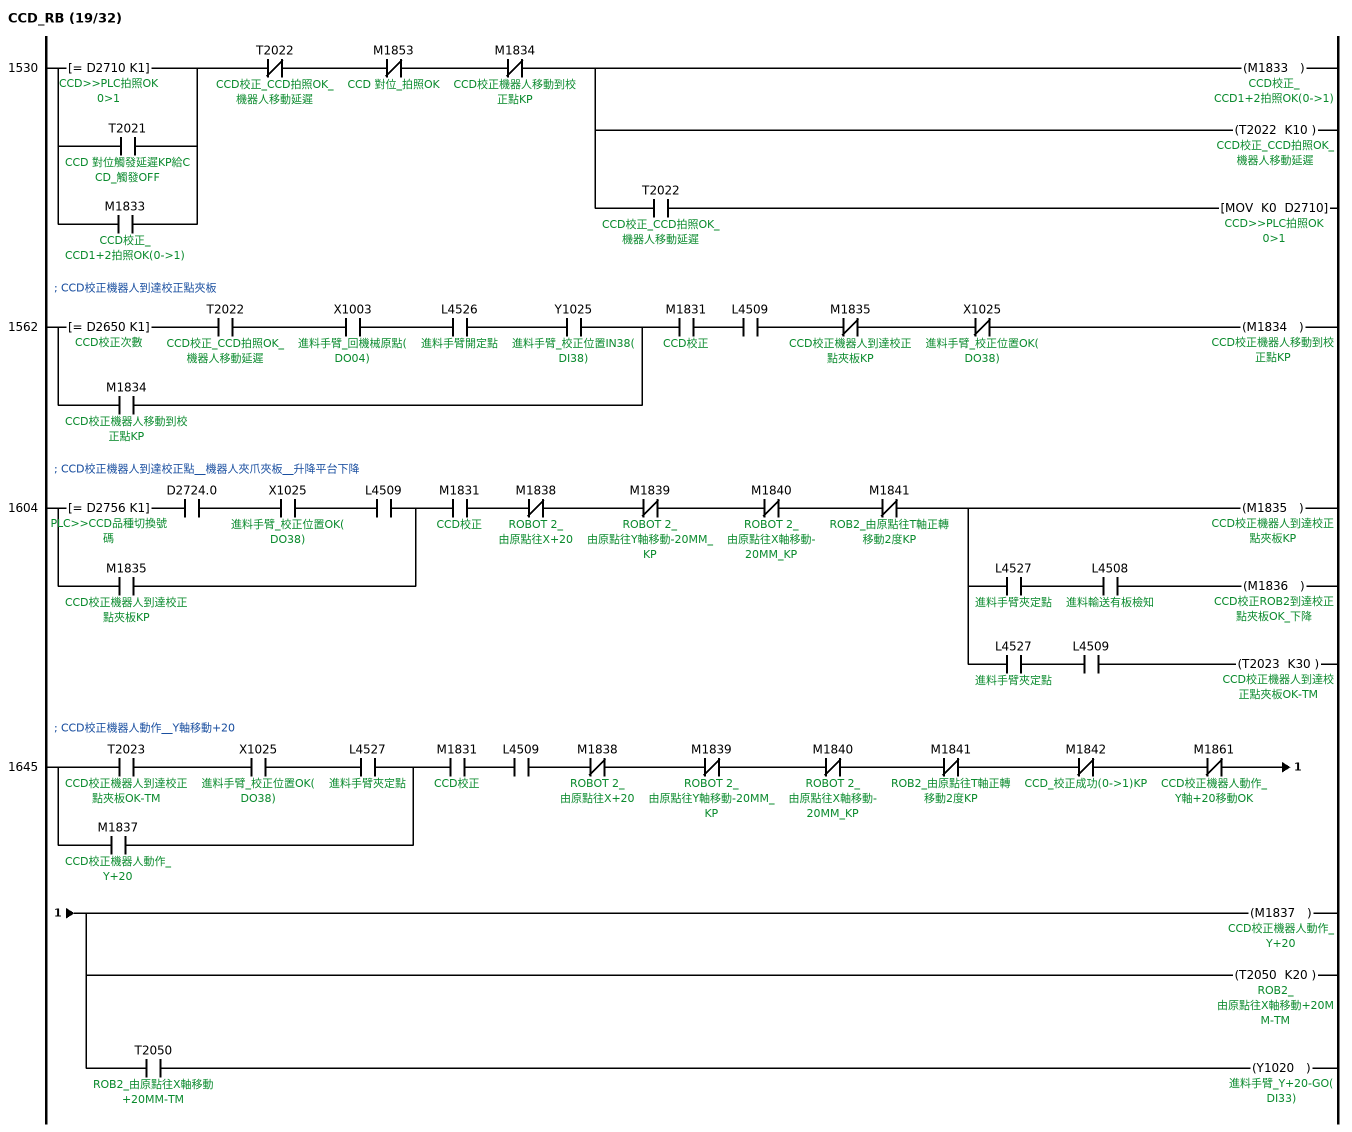
1530  LD=     D2710 K1  ; CCD>>PLC拍照OK  0>1
      OR      T2021  ; CCD 對位觸發延遲KP給CCD_觸發OFF
      OR      M1833  ; CCD校正_CCD1+2拍照OK(0->1)
      ANI     T2022  ; CCD校正_CCD拍照OK_機器人移動延遲
      ANI     M1853  ; CCD 對位_拍照OK
      ANI     M1834  ; CCD校正機器人移動到校正點KP
      OUT     M1833  ; CCD校正_CCD1+2拍照OK(0->1)
      OUT     T2022 K10  ; CCD校正_CCD拍照OK_機器人移動延遲
      AND     T2022  ; CCD校正_CCD拍照OK_機器人移動延遲
      MOV     K0 D2710
; CCD校正機器人到達校正點夾板
1562  LD=     D2650 K1  ; CCD校正次數
      AND     T2022  ; CCD校正_CCD拍照OK_機器人移動延遲
      AND     X1003  ; 進料手臂_回機械原點(DO04)
      AND     L4526  ; 進料手臂開定點
      AND     Y1025  ; 進料手臂_校正位置IN38(DI38)
      OR      M1834  ; CCD校正機器人移動到校正點KP
      AND     M1831  ; CCD校正
      AND     L4509
      ANI     M1835  ; CCD校正機器人到達校正點夾板KP
      ANI     X1025  ; 進料手臂_校正位置OK(DO38)
      OUT     M1834  ; CCD校正機器人移動到校正點KP
; CCD校正機器人到達校正點__機器人夾爪夾板__升降平台下降
1604  LD=     D2756 K1  ; PLC>>CCD品種切換號碼
      AND     D2724.0
      AND     X1025  ; 進料手臂_校正位置OK(DO38)
      AND     L4509
      OR      M1835  ; CCD校正機器人到達校正點夾板KP
      AND     M1831  ; CCD校正
      ANI     M1838  ; ROBOT 2_由原點往X+20
      ANI     M1839  ; ROBOT 2_由原點往Y軸移動-20MM_KP
      ANI     M1840  ; ROBOT 2_由原點往X軸移動-20MM_KP
      ANI     M1841  ; ROB2_由原點往T軸正轉移動2度KP
      OUT     M1835  ; CCD校正機器人到達校正點夾板KP
      MPS
      AND     L4527  ; 進料手臂夾定點
      AND     L4508  ; 進料輸送有板檢知
      OUT     M1836  ; CCD校正ROB2到達校正點夾板OK_下降
      MPP
      AND     L4527  ; 進料手臂夾定點
      AND     L4509
      OUT     T2023 K30  ; CCD校正機器人到達校正點夾板OK-TM
; CCD校正機器人動作__Y軸移動+20
1645  LD      T2023  ; CCD校正機器人到達校正點夾板OK-TM
      AND     X1025  ; 進料手臂_校正位置OK(DO38)
      AND     L4527  ; 進料手臂夾定點
      OR      M1837  ; CCD校正機器人動作_Y+20
      AND     M1831  ; CCD校正
      AND     L4509
      ANI     M1838  ; ROBOT 2_由原點往X+20
      ANI     M1839  ; ROBOT 2_由原點往Y軸移動-20MM_KP
      ANI     M1840  ; ROBOT 2_由原點往X軸移動-20MM_KP
      ANI     M1841  ; ROB2_由原點往T軸正轉移動2度KP
      ANI     M1842  ; CCD_校正成功(0->1)KP
      ANI     M1861  ; CCD校正機器人動作_Y軸+20移動OK
      OUT     M1837  ; CCD校正機器人動作_Y+20
      OUT     T2050 K20  ; ROB2_由原點往X軸移動+20MM-TM
      AND     T2050  ; ROB2_由原點往X軸移動+20MM-TM
      OUT     Y1020  ; 進料手臂_Y+20-GO(DI33)
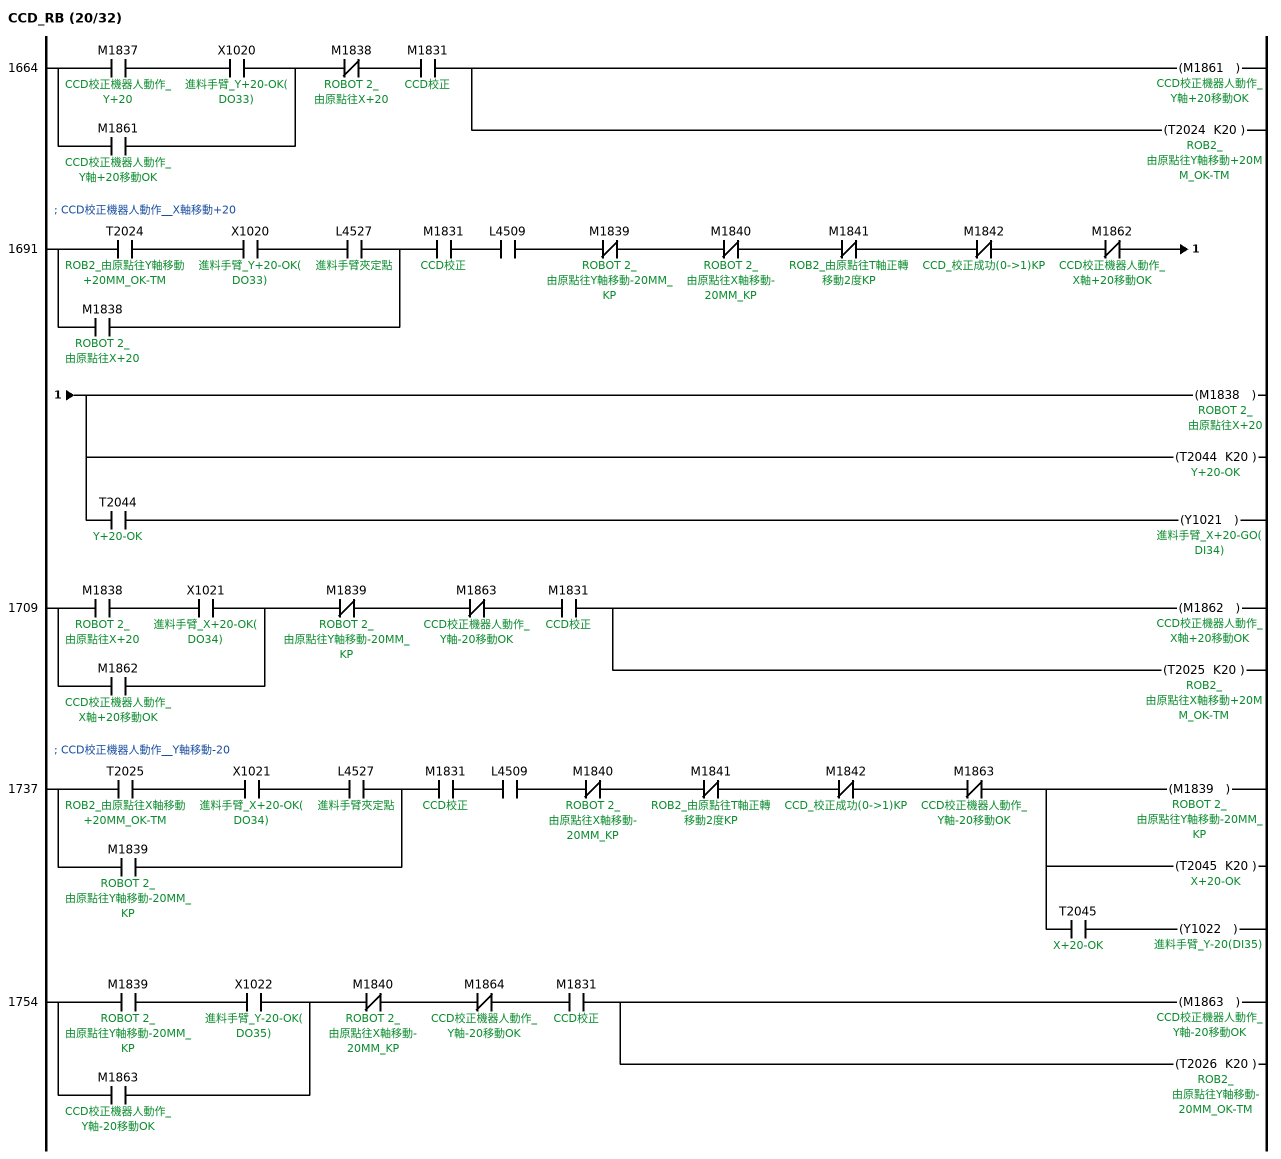
1664  LD      M1837  ; CCD校正機器人動作_Y+20
      AND     X1020  ; 進料手臂_Y+20-OK(DO33)
      OR      M1861  ; CCD校正機器人動作_Y軸+20移動OK
      ANI     M1838  ; ROBOT 2_由原點往X+20
      AND     M1831  ; CCD校正
      OUT     M1861  ; CCD校正機器人動作_Y軸+20移動OK
      OUT     T2024 K20  ; ROB2_由原點往Y軸移動+20MM_OK-TM
; CCD校正機器人動作__X軸移動+20
1691  LD      T2024  ; ROB2_由原點往Y軸移動+20MM_OK-TM
      AND     X1020  ; 進料手臂_Y+20-OK(DO33)
      AND     L4527  ; 進料手臂夾定點
      OR      M1838  ; ROBOT 2_由原點往X+20
      AND     M1831  ; CCD校正
      AND     L4509
      ANI     M1839  ; ROBOT 2_由原點往Y軸移動-20MM_KP
      ANI     M1840  ; ROBOT 2_由原點往X軸移動-20MM_KP
      ANI     M1841  ; ROB2_由原點往T軸正轉移動2度KP
      ANI     M1842  ; CCD_校正成功(0->1)KP
      ANI     M1862  ; CCD校正機器人動作_X軸+20移動OK
      OUT     M1838  ; ROBOT 2_由原點往X+20
      OUT     T2044 K20  ; Y+20-OK
      AND     T2044  ; Y+20-OK
      OUT     Y1021  ; 進料手臂_X+20-GO(DI34)
1709  LD      M1838  ; ROBOT 2_由原點往X+20
      AND     X1021  ; 進料手臂_X+20-OK(DO34)
      OR      M1862  ; CCD校正機器人動作_X軸+20移動OK
      ANI     M1839  ; ROBOT 2_由原點往Y軸移動-20MM_KP
      ANI     M1863  ; CCD校正機器人動作_Y軸-20移動OK
      AND     M1831  ; CCD校正
      OUT     M1862  ; CCD校正機器人動作_X軸+20移動OK
      OUT     T2025 K20  ; ROB2_由原點往X軸移動+20MM_OK-TM
; CCD校正機器人動作__Y軸移動-20
1737  LD      T2025  ; ROB2_由原點往X軸移動+20MM_OK-TM
      AND     X1021  ; 進料手臂_X+20-OK(DO34)
      AND     L4527  ; 進料手臂夾定點
      OR      M1839  ; ROBOT 2_由原點往Y軸移動-20MM_KP
      AND     M1831  ; CCD校正
      AND     L4509
      ANI     M1840  ; ROBOT 2_由原點往X軸移動-20MM_KP
      ANI     M1841  ; ROB2_由原點往T軸正轉移動2度KP
      ANI     M1842  ; CCD_校正成功(0->1)KP
      ANI     M1863  ; CCD校正機器人動作_Y軸-20移動OK
      OUT     M1839  ; ROBOT 2_由原點往Y軸移動-20MM_KP
      OUT     T2045 K20  ; X+20-OK
      AND     T2045  ; X+20-OK
      OUT     Y1022  ; 進料手臂_Y-20(DI35)
1754  LD      M1839  ; ROBOT 2_由原點往Y軸移動-20MM_KP
      AND     X1022  ; 進料手臂_Y-20-OK(DO35)
      OR      M1863  ; CCD校正機器人動作_Y軸-20移動OK
      ANI     M1840  ; ROBOT 2_由原點往X軸移動-20MM_KP
      ANI     M1864  ; CCD校正機器人動作_Y軸-20移動OK
      AND     M1831  ; CCD校正
      OUT     M1863  ; CCD校正機器人動作_Y軸-20移動OK
      OUT     T2026 K20  ; ROB2_由原點往Y軸移動-20MM_OK-TM
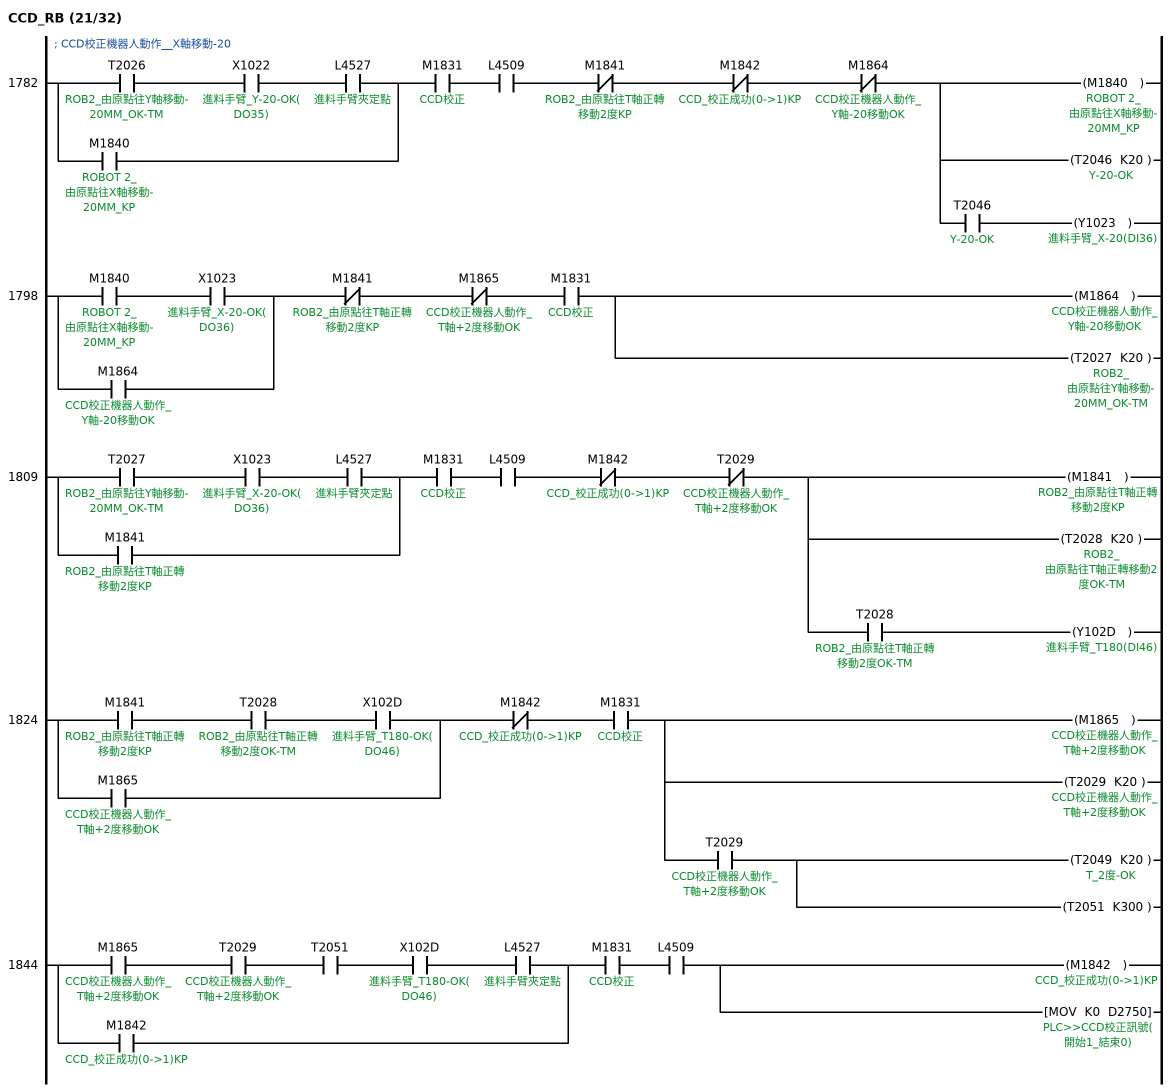
; CCD校正機器人動作__X軸移動-20
1782  LD      T2026  ; ROB2_由原點往Y軸移動-20MM_OK-TM
      AND     X1022  ; 進料手臂_Y-20-OK(DO35)
      AND     L4527  ; 進料手臂夾定點
      OR      M1840  ; ROBOT 2_由原點往X軸移動-20MM_KP
      AND     M1831  ; CCD校正
      AND     L4509
      ANI     M1841  ; ROB2_由原點往T軸正轉移動2度KP
      ANI     M1842  ; CCD_校正成功(0->1)KP
      ANI     M1864  ; CCD校正機器人動作_Y軸-20移動OK
      OUT     M1840  ; ROBOT 2_由原點往X軸移動-20MM_KP
      OUT     T2046 K20  ; Y-20-OK
      AND     T2046  ; Y-20-OK
      OUT     Y1023  ; 進料手臂_X-20(DI36)
1798  LD      M1840  ; ROBOT 2_由原點往X軸移動-20MM_KP
      AND     X1023  ; 進料手臂_X-20-OK(DO36)
      OR      M1864  ; CCD校正機器人動作_Y軸-20移動OK
      ANI     M1841  ; ROB2_由原點往T軸正轉移動2度KP
      ANI     M1865  ; CCD校正機器人動作_T軸+2度移動OK
      AND     M1831  ; CCD校正
      OUT     M1864  ; CCD校正機器人動作_Y軸-20移動OK
      OUT     T2027 K20  ; ROB2_由原點往Y軸移動-20MM_OK-TM
1809  LD      T2027  ; ROB2_由原點往Y軸移動-20MM_OK-TM
      AND     X1023  ; 進料手臂_X-20-OK(DO36)
      AND     L4527  ; 進料手臂夾定點
      OR      M1841  ; ROB2_由原點往T軸正轉移動2度KP
      AND     M1831  ; CCD校正
      AND     L4509
      ANI     M1842  ; CCD_校正成功(0->1)KP
      ANI     T2029  ; CCD校正機器人動作_T軸+2度移動OK
      OUT     M1841  ; ROB2_由原點往T軸正轉移動2度KP
      OUT     T2028 K20  ; ROB2_由原點往T軸正轉移動2度OK-TM
      AND     T2028  ; ROB2_由原點往T軸正轉移動2度OK-TM
      OUT     Y102D  ; 進料手臂_T180(DI46)
1824  LD      M1841  ; ROB2_由原點往T軸正轉移動2度KP
      AND     T2028  ; ROB2_由原點往T軸正轉移動2度OK-TM
      AND     X102D  ; 進料手臂_T180-OK(DO46)
      OR      M1865  ; CCD校正機器人動作_T軸+2度移動OK
      ANI     M1842  ; CCD_校正成功(0->1)KP
      AND     M1831  ; CCD校正
      OUT     M1865  ; CCD校正機器人動作_T軸+2度移動OK
      OUT     T2029 K20  ; CCD校正機器人動作_T軸+2度移動OK
      AND     T2029  ; CCD校正機器人動作_T軸+2度移動OK
      OUT     T2049 K20  ; T_2度-OK
      OUT     T2051 K300
1844  LD      M1865  ; CCD校正機器人動作_T軸+2度移動OK
      AND     T2029  ; CCD校正機器人動作_T軸+2度移動OK
      AND     T2051
      AND     X102D  ; 進料手臂_T180-OK(DO46)
      AND     L4527  ; 進料手臂夾定點
      OR      M1842  ; CCD_校正成功(0->1)KP
      AND     M1831  ; CCD校正
      AND     L4509
      OUT     M1842  ; CCD_校正成功(0->1)KP
      MOV     K0 D2750
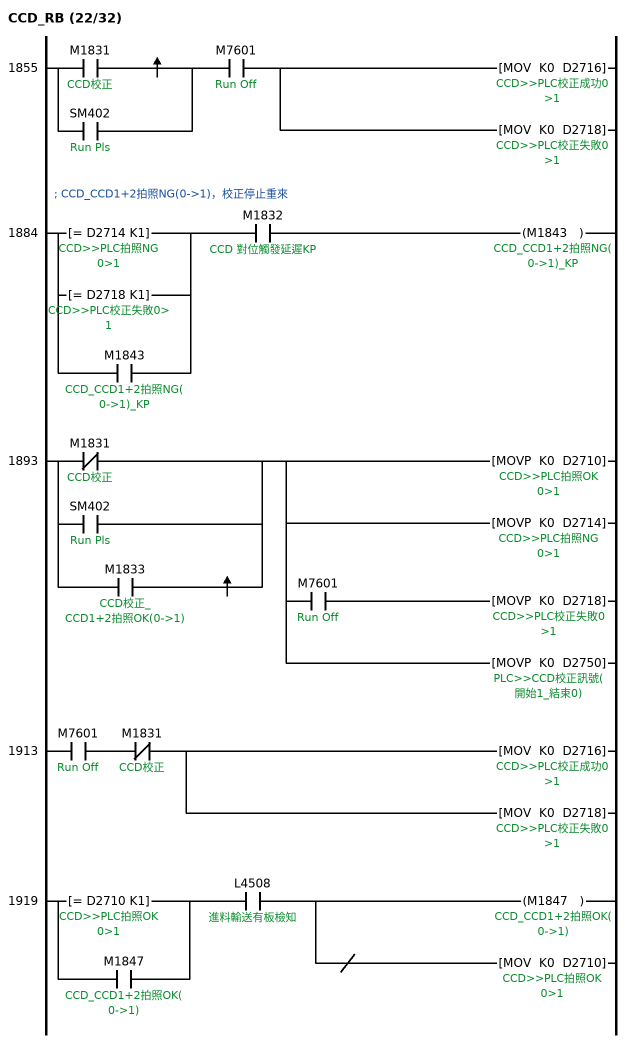
1855  LD      M1831  ; CCD校正
      MEP
      OR      SM402  ; Run Pls
      AND     M7601  ; Run Off
      MOV     K0 D2716  ; CCD>>PLC校正成功0>1
      MOV     K0 D2718  ; CCD>>PLC校正失敗0>1
; CCD_CCD1+2拍照NG(0->1)，校正停止重來
1884  LD=     D2714 K1  ; CCD>>PLC拍照NG  0>1
      OR=     D2718 K1  ; CCD>>PLC校正失敗0>1
      OR      M1843  ; CCD_CCD1+2拍照NG(0->1)_KP
      AND     M1832  ; CCD 對位觸發延遲KP
      OUT     M1843  ; CCD_CCD1+2拍照NG(0->1)_KP
1893  LDI     M1831  ; CCD校正
      OR      SM402  ; Run Pls
      LD      M1833  ; CCD校正_CCD1+2拍照OK(0->1)
      MEP
      ORB
      MOVP    K0 D2710
      MOVP    K0 D2714
      MPS
      AND     M7601  ; Run Off
      MOVP    K0 D2718
      MPP
      MOVP    K0 D2750
1913  LD      M7601  ; Run Off
      ANI     M1831  ; CCD校正
      MOV     K0 D2716
      MOV     K0 D2718
1919  LD=     D2710 K1  ; CCD>>PLC拍照OK  0>1
      OR      M1847  ; CCD_CCD1+2拍照OK(0->1)
      AND     L4508  ; 進料輸送有板檢知
      OUT     M1847  ; CCD_CCD1+2拍照OK(0->1)
      INV
      MOV     K0 D2710
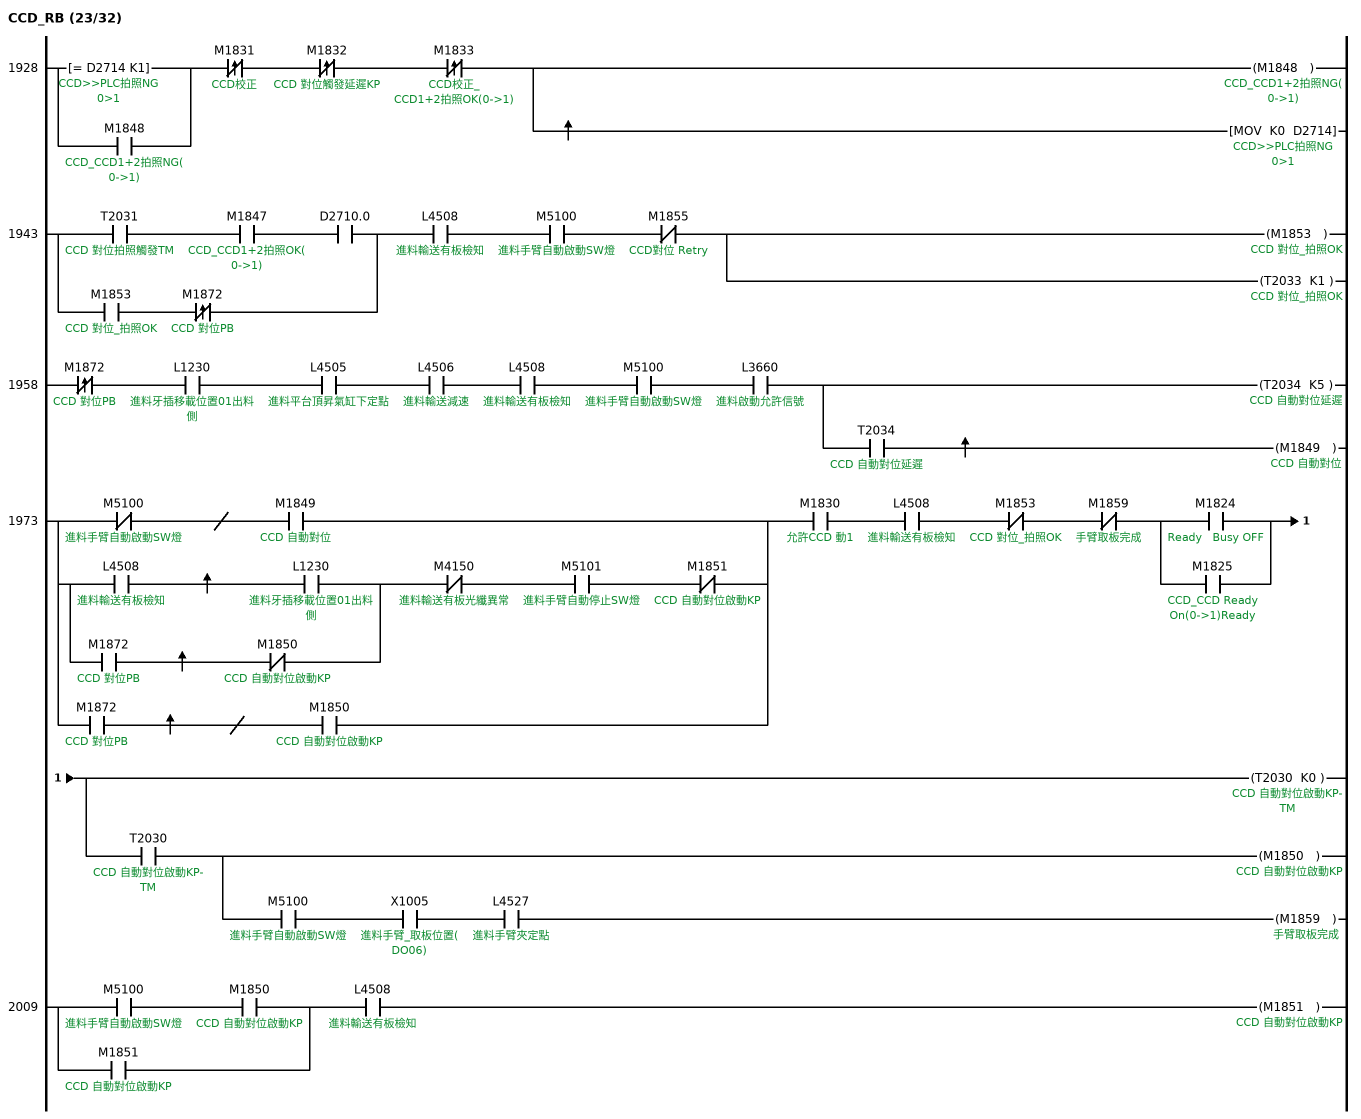
1928  LD=     D2714 K1  ; CCD>>PLC拍照NG  0>1
      OR      M1848  ; CCD_CCD1+2拍照NG(0->1)
      ANDPI   M1831  ; CCD校正
      ANDPI   M1832  ; CCD 對位觸發延遲KP
      ANDPI   M1833  ; CCD校正_CCD1+2拍照OK(0->1)
      OUT     M1848  ; CCD_CCD1+2拍照NG(0->1)
      MEP
      MOV     K0 D2714
1943  LD      T2031  ; CCD 對位拍照觸發TM
      AND     M1847  ; CCD_CCD1+2拍照OK(0->1)
      AND     D2710.0
      LD      M1853  ; CCD 對位_拍照OK
      ANDPI   M1872  ; CCD 對位PB
      ORB
      AND     L4508  ; 進料輸送有板檢知
      AND     M5100  ; 進料手臂自動啟動SW燈
      ANI     M1855  ; CCD對位 Retry
      OUT     M1853  ; CCD 對位_拍照OK
      OUT     T2033 K1  ; CCD 對位_拍照OK
1958  LDPI    M1872  ; CCD 對位PB
      AND     L1230  ; 進料牙插移載位置01出料側
      AND     L4505  ; 進料平台頂昇氣缸下定點
      AND     L4506  ; 進料輸送減速
      AND     L4508  ; 進料輸送有板檢知
      AND     M5100  ; 進料手臂自動啟動SW燈
      AND     L3660  ; 進料啟動允許信號
      OUT     T2034 K5  ; CCD 自動對位延遲
      AND     T2034  ; CCD 自動對位延遲
      MEP
      OUT     M1849  ; CCD 自動對位
1973  LDI     M5100  ; 進料手臂自動啟動SW燈
      INV
      AND     M1849  ; CCD 自動對位
      LD      L4508  ; 進料輸送有板檢知
      MEP
      AND     L1230  ; 進料牙插移載位置01出料側
      LD      M1872  ; CCD 對位PB
      MEP
      ANI     M1850  ; CCD 自動對位啟動KP
      ORB
      ANI     M4150  ; 進料輸送有板光纖異常
      AND     M5101  ; 進料手臂自動停止SW燈
      ANI     M1851  ; CCD 自動對位啟動KP
      ORB
      LD      M1872  ; CCD 對位PB
      MEP
      INV
      AND     M1850  ; CCD 自動對位啟動KP
      ORB
      AND     M1830  ; 允許CCD 動1
      AND     L4508  ; 進料輸送有板檢知
      ANI     M1853  ; CCD 對位_拍照OK
      ANI     M1859  ; 手臂取板完成
      LD      M1824  ; Ready   Busy OFF
      OR      M1825  ; CCD_CCD Ready On(0->1)Ready
      ANB
      OUT     T2030 K0  ; CCD 自動對位啟動KP-TM
      AND     T2030  ; CCD 自動對位啟動KP-TM
      OUT     M1850  ; CCD 自動對位啟動KP
      AND     M5100  ; 進料手臂自動啟動SW燈
      AND     X1005  ; 進料手臂_取板位置(DO06)
      AND     L4527  ; 進料手臂夾定點
      OUT     M1859  ; 手臂取板完成
2009  LD      M5100  ; 進料手臂自動啟動SW燈
      AND     M1850  ; CCD 自動對位啟動KP
      OR      M1851  ; CCD 自動對位啟動KP
      AND     L4508  ; 進料輸送有板檢知
      OUT     M1851  ; CCD 自動對位啟動KP
